// TwinCAT 3 PLC project Sorting_Machine_PLC
// ProgramVersion: 3.1.4024.0
// libraries:
//   Tc2_MC2, * (Beckhoff Automation GmbH)
//   Tc2_Standard, * (Beckhoff Automation GmbH)
//   Tc2_System, * (Beckhoff Automation GmbH)
//   Tc3_Module, * (Beckhoff Automation GmbH)
// project tree:
//   00_Internal PackML/DUTs/ E_PMLState.TcDUT, E_PMLUnitMode.TcDUT
//   00_Internal PackML/POUs/ PS_PackML_StateMachine_Auto.TcPOU, PS_PackML_StateMachine_Maintenance.TcPOU, PS_PackML_StateMachine_Manual.TcPOU, PS_PackML_StateMachine_SemiAuto.TcPOU, PS_PackML_UnitModeManager.TcPOU
//   01_Submodules/Axis/ FB_Axis.TcPOU
//   01_Submodules/Cylinder/ FB_CylinderDiag.TcPOU, FB_CylinderTemp.TcPOU, FB_CylinderTempDiag.TcPOU, FB_CylinderTempRecord.TcPOU, I_Cylinder.TcIO, FB_CylinderBase.TcPOU
//   01_Submodules/Sensor %28signal handling%29/ FB_SignalHandling.TcPOU (not stored), FB_SignalHandlingIntern.TcPOU (not stored), I_SignalHandling.TcIO (not stored), FB_SignalHandlingDelay.TcPOU (not stored)
//   02_Subsystems/ E_StateSeparatingAutoClampBarrier.TcDUT, E_StateSortingAutoAxis.TcDUT, E_StateSortingAutoCylinder.TcDUT, FB_SeparatingModule.TcPOU, FB_SortingModule.TcPOU, FB_SubsystemRoot.TcPOU
//   03_Machine/ FB_Machine.TcPOU
//   / PlcTask.TcTTO
//   04_Application/ MAIN.TcPOU
// real-time tasks:
//   TASK PlcTask: cycle T#10ms, priority 20, ADS port 350

CONFIGURATION Sorting_Machine_PLC
    RESOURCE PLC ON TwinCAT3
        TASK PlcTask(INTERVAL := T#10ms, PRIORITY := 20);
        PROGRAM MAIN WITH PlcTask : MAIN;
    END_RESOURCE
END_CONFIGURATION

// ---- 00_Internal PackML/DUTs/E_PMLState.TcDUT
{attribute 'qualified_only'}
{attribute 'strict'}
TYPE E_PMLState :
(
	UNDEFINED 			:=	0,
	CLEARING			:=	1,
	STOPPED				:=	2,
	STARTING			:=	3,
	IDLE				:=	4,
	SUSPENDED			:=	5,
	EXECUTE				:=	6,
	STOPPING			:=	7,
	ABORTING			:=	8,
	ABORTED				:=	9,
	HOLDING				:=	10,
	HELD				:=	11,
	UNHOLDING			:=	12,
	SUSPENDING			:=	13,
	UNSUSPENDING		:=	14,
	RESETTING			:=	15,
	COMPLETING			:=	16,
	COMPLETE			:=	17
);
END_TYPE

// ---- 00_Internal PackML/DUTs/E_PMLUnitMode.TcDUT
{attribute 'qualified_only'}
{attribute 'strict'}
TYPE E_PMLUnitMode :
(
	UNDEFINED 			:=	0,
	AUTOMATIC			:=	1,
	MAINTENANCE			:=	2,
	MANUAL				:=	3,
	SEMIAUTOMATIC		:=	4,
	DRYRUN				:=	5,
	USERMODE1			:=	6,
	USERMODE2			:=	7,
	IDLE				:=	8,
	ESTOP				:=	9
);
END_TYPE

// ---- 02_Subsystems/E_StateSeparatingAutoClampBarrier.TcDUT
{attribute 'qualified_only'}
{attribute 'strict'}
TYPE E_StateSeparatingAutoClampBarrier :
(
	Init 			:= 0,
	Start,
	CloseClamp,
	OpenBarrier,
	CloseBarrier,
	OpenClamp
);
END_TYPE

// ---- 02_Subsystems/E_StateSortingAutoAxis.TcDUT
{attribute 'qualified_only'}
{attribute 'strict'}
TYPE E_StateSortingAutoAxis :
(
	WaitForCylinderAtWorkPos 			:= 0,
	MoveAxis,
	StopAxis
);
END_TYPE

// ---- 02_Subsystems/E_StateSortingAutoCylinder.TcDUT
{attribute 'qualified_only'}
{attribute 'strict'}
TYPE E_StateSortingAutoCylinder :
(
	BoxDetected 			:= 0,
	MoveCylToWorkPos,
	MoveCylToBasePos
);
END_TYPE

// ---- 01_Submodules/Cylinder/I_Cylinder.TcIO
INTERFACE I_Cylinder

PROPERTY bState_AtBasePos : BOOL
GET
END_GET
END_PROPERTY

PROPERTY bState_AtWorkPos : BOOL
GET
END_GET
END_PROPERTY

PROPERTY bState_MoveToWork : BOOL
GET
END_GET
END_PROPERTY

METHOD MoveToBase
VAR_INPUT
END_VAR
END_METHOD

METHOD MoveToWork
VAR_INPUT
END_VAR
END_METHOD

METHOD Reset
VAR_INPUT
END_VAR
END_METHOD

END_INTERFACE

// ---- 04_Application/MAIN.TcPOU
PROGRAM MAIN
VAR
END_VAR

END_PROGRAM

// ---- 00_Internal PackML/POUs/PS_PackML_StateMachine_Auto.TcPOU
FUNCTION_BLOCK PS_PackML_StateMachine_Auto
VAR_INPUT
	Start					:	BOOL;
	Hold					:	BOOL;
	UnHold					:	BOOL;
	Suspend					:	BOOL;
	UnSuspend				:	BOOL;
	Abort					:	BOOL;
	Stop					:	BOOL;
	Complete				:	BOOL;
	Clear					:	BOOL;
	Reset					:	BOOL;
	StateComplete			:	BOOL;
END_VAR
VAR_OUTPUT
	Status					:	WORD;
	// Transient states
	ST_Starting				:	BOOL;
	ST_Completing			:	BOOL;
	ST_Resetting			:	BOOL;
	ST_Holding				:	BOOL;
	ST_UnHolding			:	BOOL;
	ST_Suspending			:	BOOL;
	ST_UnSuspending			:	BOOL;
	ST_Clearing				:	BOOL;
	ST_Stopping				:	BOOL;
	ST_Aborting				:	BOOL;
	// Final states
	ST_Execute				:	BOOL;
	ST_Complete				:	BOOL;
	ST_Idle					:	BOOL;
	ST_Held					:	BOOL;
	ST_Suspended			:	BOOL;
	ST_Stopped				:	BOOL;
	ST_Aborted				:	BOOL;
	
	Error					:	BOOL;
	ErrorID					:	DWORD;
	ePMLState				:	E_PMLState	:=	E_PMLState.IDLE;
END_VAR
VAR
	ePMLStatePrev			:	E_PMLState;
	bStateChange			:	BOOL;
	bStateCompletePrev		:	BOOL;
END_VAR

	// Check for E_PMLState change
	IF ePMLStatePrev <> ePMLState THEN
		ePMLStatePrev	:=	ePMLState;
		bStateChange	:=	TRUE;
	ELSE
		bStateChange	:=	FALSE;
	END_IF
	
	// change to new state if requested
	CASE ePMLState OF
		E_PMLState.UNDEFINED:
			IF bStateChange	THEN
				ST_Starting				:=	FALSE;
				ST_Completing			:=	FALSE;
				ST_Resetting			:=	FALSE;
				ST_Holding				:=	FALSE;
				ST_UnHolding			:=	FALSE;
				ST_Suspending			:=	FALSE;
				ST_UnSuspending			:=	FALSE;
				ST_Clearing				:=	FALSE;
				ST_Stopping				:=	FALSE;
				ST_Aborting				:=	FALSE;
				
				ST_Execute				:=	FALSE;
				ST_Complete				:=	FALSE;
				ST_Idle					:=	FALSE;
				ST_Held					:=	FALSE;
				ST_Suspended			:=	FALSE;
				ST_Stopped				:=	FALSE;
				ST_Aborted				:=	FALSE;
			END_IF
			
			IF Abort THEN
				ePMLState				:=	E_PMLState.ABORTING;
				ST_Aborting				:=	TRUE;
			ELSIF Stop THEN
				ePMLState				:=	E_PMLState.STOPPING;
				ST_Stopping				:=	TRUE;				
			END_IF
		
		E_PMLState.IDLE:
			IF bStateChange	THEN
				ST_Starting				:=	FALSE;
				ST_Completing			:=	FALSE;
				ST_Resetting			:=	FALSE;
				ST_Holding				:=	FALSE;
				ST_UnHolding			:=	FALSE;
				ST_Suspending			:=	FALSE;
				ST_UnSuspending			:=	FALSE;
				ST_Clearing				:=	FALSE;
				ST_Stopping				:=	FALSE;
				ST_Aborting				:=	FALSE;
				
				ST_Execute				:=	FALSE;
				ST_Complete				:=	FALSE;
				ST_Idle					:=	TRUE;
				ST_Held					:=	FALSE;
				ST_Suspended			:=	FALSE;
				ST_Stopped				:=	FALSE;
				ST_Aborted				:=	FALSE;
			END_IF
			
			IF Abort THEN
				ePMLState				:=	E_PMLState.ABORTING;
				ST_IDLE					:=	FALSE;
				ST_Aborting				:=	TRUE;
			ELSIF Stop THEN
				ePMLState				:=	E_PMLState.STOPPING;
				ST_IDLE					:=	FALSE;
				ST_Stopping				:=	TRUE;
			ELSIF Start THEN
				ePMLState				:=	E_PMLState.STARTING;
				ST_IDLE					:=	FALSE;
				ST_Starting				:=	TRUE;								
			END_IF

		E_PMLState.STARTING:
			IF bStateChange	THEN
				ST_Starting				:=	TRUE;
				ST_Completing			:=	FALSE;
				ST_Resetting			:=	FALSE;
				ST_Holding				:=	FALSE;
				ST_UnHolding			:=	FALSE;
				ST_Suspending			:=	FALSE;
				ST_UnSuspending			:=	FALSE;
				ST_Clearing				:=	FALSE;
				ST_Stopping				:=	FALSE;
				ST_Aborting				:=	FALSE;
				
				ST_Execute				:=	FALSE;
				ST_Complete				:=	FALSE;
				ST_Idle					:=	FALSE;
				ST_Held					:=	FALSE;
				ST_Suspended			:=	FALSE;
				ST_Stopped				:=	FALSE;
				ST_Aborted				:=	FALSE;
			END_IF
			
			IF Abort THEN
				ePMLState				:=	E_PMLState.ABORTING;
				ST_Starting				:=	FALSE;
				ST_Aborting				:=	TRUE;
			ELSIF Stop THEN
				ePMLState				:=	E_PMLState.STOPPING;
				ST_Starting				:=	FALSE;
				ST_Stopping				:=	TRUE;
			ELSIF StateComplete AND NOT bStateCompletePrev THEN
				ePMLState				:=	E_PMLState.EXECUTE;
				bStateCompletePrev		:=	StateComplete;
				ST_Starting				:=	FALSE;
				ST_Execute				:=	TRUE;								
			END_IF

		E_PMLState.EXECUTE:
			IF bStateChange	THEN
				ST_Starting				:=	FALSE;
				ST_Completing			:=	FALSE;
				ST_Resetting			:=	FALSE;
				ST_Holding				:=	FALSE;
				ST_UnHolding			:=	FALSE;
				ST_Suspending			:=	FALSE;
				ST_UnSuspending			:=	FALSE;
				ST_Clearing				:=	FALSE;
				ST_Stopping				:=	FALSE;
				ST_Aborting				:=	FALSE;
				
				ST_Execute				:=	TRUE;
				ST_Complete				:=	FALSE;
				ST_Idle					:=	FALSE;
				ST_Held					:=	FALSE;
				ST_Suspended			:=	FALSE;
				ST_Stopped				:=	FALSE;
				ST_Aborted				:=	FALSE;
			END_IF
			
			IF Abort THEN
				ePMLState				:=	E_PMLState.ABORTING;
				ST_Execute				:=	FALSE;
				ST_Aborting				:=	TRUE;
			ELSIF Stop THEN
				ePMLState				:=	E_PMLState.STOPPING;
				ST_Execute				:=	FALSE;
				ST_Stopping				:=	TRUE;
			ELSIF Hold THEN
				ePMLState				:=	E_PMLState.HOLDING;
				ST_Execute				:=	FALSE;
				ST_Holding				:=	TRUE;
			ELSIF Suspend THEN
				ePMLState				:=	E_PMLState.SUSPENDING;
				ST_Execute				:=	FALSE;
				ST_Suspending			:=	TRUE;
			ELSIF Complete THEN
				ePMLState				:=	E_PMLState.COMPLETING;
				ST_Execute				:=	FALSE;
				ST_Completing			:=	TRUE;	
			END_IF

		E_PMLState.COMPLETING:
			IF bStateChange	THEN
				ST_Starting				:=	FALSE;
				ST_Completing			:=	TRUE;
				ST_Resetting			:=	FALSE;
				ST_Holding				:=	FALSE;
				ST_UnHolding			:=	FALSE;
				ST_Suspending			:=	FALSE;
				ST_UnSuspending			:=	FALSE;
				ST_Clearing				:=	FALSE;
				ST_Stopping				:=	FALSE;
				ST_Aborting				:=	FALSE;
				
				ST_Execute				:=	FALSE;
				ST_Complete				:=	FALSE;
				ST_Idle					:=	FALSE;
				ST_Held					:=	FALSE;
				ST_Suspended			:=	FALSE;
				ST_Stopped				:=	FALSE;
				ST_Aborted				:=	FALSE;
			END_IF
			
			IF Abort THEN
				ePMLState				:=	E_PMLState.ABORTING;
				ST_Completing			:=	FALSE;
				ST_Aborting				:=	TRUE;
			ELSIF Stop THEN
				ePMLState				:=	E_PMLState.STOPPING;
				ST_Completing			:=	FALSE;
				ST_Stopping				:=	TRUE;
			ELSIF StateComplete AND NOT bStateCompletePrev THEN
				ePMLState				:=	E_PMLState.COMPLETE;
				bStateCompletePrev		:=	StateComplete;
				ST_Completing			:=	FALSE;
				ST_Complete				:=	TRUE;								
			END_IF
			
		E_PMLState.COMPLETE:
			IF bStateChange	THEN
				ST_Starting				:=	FALSE;
				ST_Completing			:=	FALSE;
				ST_Resetting			:=	FALSE;
				ST_Holding				:=	FALSE;
				ST_UnHolding			:=	FALSE;
				ST_Suspending			:=	FALSE;
				ST_UnSuspending			:=	FALSE;
				ST_Clearing				:=	FALSE;
				ST_Stopping				:=	FALSE;
				ST_Aborting				:=	FALSE;
				
				ST_Execute				:=	FALSE;
				ST_Complete				:=	TRUE;
				ST_Idle					:=	FALSE;
				ST_Held					:=	FALSE;
				ST_Suspended			:=	FALSE;
				ST_Stopped				:=	FALSE;
				ST_Aborted				:=	FALSE;
			END_IF
			
			IF Abort THEN
				ePMLState				:=	E_PMLState.ABORTING;
				ST_Complete				:=	FALSE;
				ST_Aborting				:=	TRUE;
			ELSIF Stop THEN
				ePMLState				:=	E_PMLState.STOPPING;
				ST_Complete				:=	FALSE;
				ST_Stopping				:=	TRUE;
			ELSIF Reset THEN
				ePMLState				:=	E_PMLState.RESETTING;
				ST_Complete				:=	FALSE;
				ST_Resetting			:=	TRUE;
			END_IF

		E_PMLState.RESETTING:
			IF bStateChange	THEN
				ST_Starting				:=	FALSE;
				ST_Completing			:=	FALSE;
				ST_Resetting			:=	TRUE;
				ST_Holding				:=	FALSE;
				ST_UnHolding			:=	FALSE;
				ST_Suspending			:=	FALSE;
				ST_UnSuspending			:=	FALSE;
				ST_Clearing				:=	FALSE;
				ST_Stopping				:=	FALSE;
				ST_Aborting				:=	FALSE;
				
				ST_Execute				:=	FALSE;
				ST_Complete				:=	FALSE;
				ST_Idle					:=	FALSE;
				ST_Held					:=	FALSE;
				ST_Suspended			:=	FALSE;
				ST_Stopped				:=	FALSE;
				ST_Aborted				:=	FALSE;
			END_IF
			
			IF Abort THEN
				ePMLState				:=	E_PMLState.ABORTING;
				ST_Resetting			:=	FALSE;
				ST_Aborting				:=	TRUE;
			ELSIF Stop THEN
				ePMLState				:=	E_PMLState.STOPPING;
				ST_Resetting			:=	FALSE;
				ST_Stopping				:=	TRUE;
			ELSIF StateComplete AND NOT bStateCompletePrev THEN
				ePMLState				:=	E_PMLState.IDLE;
				bStateCompletePrev		:=	StateComplete;
				ST_Resetting			:=	FALSE;
				ST_Idle					:=	TRUE;								
			END_IF
		
		E_PMLState.HOLDING:
			IF bStateChange	THEN
				ST_Starting				:=	FALSE;
				ST_Completing			:=	FALSE;
				ST_Resetting			:=	FALSE;
				ST_Holding				:=	TRUE;
				ST_UnHolding			:=	FALSE;
				ST_Suspending			:=	FALSE;
				ST_UnSuspending			:=	FALSE;
				ST_Clearing				:=	FALSE;
				ST_Stopping				:=	FALSE;
				ST_Aborting				:=	FALSE;
				
				ST_Execute				:=	FALSE;
				ST_Complete				:=	FALSE;
				ST_Idle					:=	FALSE;
				ST_Held					:=	FALSE;
				ST_Suspended			:=	FALSE;
				ST_Stopped				:=	FALSE;
				ST_Aborted				:=	FALSE;
			END_IF
			
			IF Abort THEN
				ePMLState				:=	E_PMLState.ABORTING;
				ST_Holding				:=	FALSE;
				ST_Aborting				:=	TRUE;
			ELSIF Stop THEN
				ePMLState				:=	E_PMLState.STOPPING;
				ST_Holding				:=	FALSE;
				ST_Stopping				:=	TRUE;
			ELSIF StateComplete AND NOT bStateCompletePrev THEN
				ePMLState				:=	E_PMLState.HELD;
				bStateCompletePrev		:=	StateComplete;
				ST_Holding				:=	FALSE;
				ST_Held					:=	TRUE;								
			END_IF
			
		E_PMLState.HELD:
			IF bStateChange	THEN
				ST_Starting				:=	FALSE;
				ST_Completing			:=	FALSE;
				ST_Resetting			:=	FALSE;
				ST_Holding				:=	FALSE;
				ST_UnHolding			:=	FALSE;
				ST_Suspending			:=	FALSE;
				ST_UnSuspending			:=	FALSE;
				ST_Clearing				:=	FALSE;
				ST_Stopping				:=	FALSE;
				ST_Aborting				:=	FALSE;
				
				ST_Execute				:=	FALSE;
				ST_Complete				:=	FALSE;
				ST_Idle					:=	FALSE;
				ST_Held					:=	TRUE;
				ST_Suspended			:=	FALSE;
				ST_Stopped				:=	FALSE;
				ST_Aborted				:=	FALSE;
			END_IF
			
			IF Abort THEN
				ePMLState				:=	E_PMLState.ABORTING;
				ST_Held					:=	FALSE;
				ST_Aborting				:=	TRUE;
			ELSIF Stop THEN
				ePMLState				:=	E_PMLState.STOPPING;
				ST_Held					:=	FALSE;
				ST_Stopping				:=	TRUE;
			ELSIF UnHold THEN
				ePMLState				:=	E_PMLState.UNHOLDING;
				ST_Held					:=	FALSE;
				ST_UnHolding			:=	TRUE;
			END_IF

		E_PMLState.UNHOLDING:	
			IF bStateChange	THEN
				ST_Starting				:=	FALSE;
				ST_Completing			:=	FALSE;
				ST_Resetting			:=	FALSE;
				ST_Holding				:=	FALSE;
				ST_UnHolding			:=	TRUE;
				ST_Suspending			:=	FALSE;
				ST_UnSuspending			:=	FALSE;
				ST_Clearing				:=	FALSE;
				ST_Stopping				:=	FALSE;
				ST_Aborting				:=	FALSE;
				
				ST_Execute				:=	FALSE;
				ST_Complete				:=	FALSE;
				ST_Idle					:=	FALSE;
				ST_Held					:=	FALSE;
				ST_Suspended			:=	FALSE;
				ST_Stopped				:=	FALSE;
				ST_Aborted				:=	FALSE;
			END_IF
			
			IF Abort THEN
				ePMLState				:=	E_PMLState.ABORTING;
				ST_UnHolding			:=	FALSE;
				ST_Aborting				:=	TRUE;
			ELSIF Stop THEN
				ePMLState				:=	E_PMLState.STOPPING;
				ST_UnHolding			:=	FALSE;
				ST_Stopping				:=	TRUE;
			ELSIF StateComplete AND NOT bStateCompletePrev THEN
				ePMLState				:=	E_PMLState.EXECUTE;
				bStateCompletePrev		:=	StateComplete;
				ST_UnHolding			:=	FALSE;
				ST_Execute				:=	TRUE;								
			END_IF
			
		E_PMLState.SUSPENDING:
			IF bStateChange	THEN
				ST_Starting				:=	FALSE;
				ST_Completing			:=	FALSE;
				ST_Resetting			:=	FALSE;
				ST_Holding				:=	FALSE;
				ST_UnHolding			:=	FALSE;
				ST_Suspending			:=	TRUE;
				ST_UnSuspending			:=	FALSE;
				ST_Clearing				:=	FALSE;
				ST_Stopping				:=	FALSE;
				ST_Aborting				:=	FALSE;
				
				ST_Execute				:=	FALSE;
				ST_Complete				:=	FALSE;
				ST_Idle					:=	FALSE;
				ST_Held					:=	FALSE;
				ST_Suspended			:=	FALSE;
				ST_Stopped				:=	FALSE;
				ST_Aborted				:=	FALSE;
			END_IF
			
			IF Abort THEN
				ePMLState				:=	E_PMLState.ABORTING;
				ST_Suspending			:=	FALSE;
				ST_Aborting				:=	TRUE;
			ELSIF Stop THEN
				ePMLState				:=	E_PMLState.STOPPING;
				ST_Suspending			:=	FALSE;
				ST_Stopping				:=	TRUE;
			ELSIF StateComplete AND NOT bStateCompletePrev THEN
				ePMLState				:=	E_PMLState.SUSPENDED;
				bStateCompletePrev		:=	StateComplete;
				ST_Suspending			:=	FALSE;
				ST_Suspended			:=	TRUE;								
			END_IF
		
		E_PMLState.SUSPENDED:
			IF bStateChange	THEN
				ST_Starting				:=	FALSE;
				ST_Completing			:=	FALSE;
				ST_Resetting			:=	FALSE;
				ST_Holding				:=	FALSE;
				ST_UnHolding			:=	FALSE;
				ST_Suspending			:=	FALSE;
				ST_UnSuspending			:=	FALSE;
				ST_Clearing				:=	FALSE;
				ST_Stopping				:=	FALSE;
				ST_Aborting				:=	FALSE;
				
				ST_Execute				:=	FALSE;
				ST_Complete				:=	FALSE;
				ST_Idle					:=	FALSE;
				ST_Held					:=	FALSE;
				ST_Suspended			:=	TRUE;
				ST_Stopped				:=	FALSE;
				ST_Aborted				:=	FALSE;
			END_IF
			
			IF Abort THEN
				ePMLState				:=	E_PMLState.ABORTING;
				ST_Suspended			:=	FALSE;
				ST_Aborting				:=	TRUE;
			ELSIF Stop THEN
				ePMLState				:=	E_PMLState.STOPPING;
				ST_Suspended			:=	FALSE;
				ST_Stopping				:=	TRUE;
			ELSIF UnSuspend THEN
				ePMLState				:=	E_PMLState.UNSUSPENDING;
				ST_Suspended			:=	FALSE;
				ST_UnSuspending			:=	TRUE;
			END_IF

		E_PMLState.UNSUSPENDING:	
			IF bStateChange	THEN
				ST_Starting				:=	FALSE;
				ST_Completing			:=	FALSE;
				ST_Resetting			:=	FALSE;
				ST_Holding				:=	FALSE;
				ST_UnHolding			:=	FALSE;
				ST_Suspending			:=	FALSE;
				ST_UnSuspending			:=	TRUE;
				ST_Clearing				:=	FALSE;
				ST_Stopping				:=	FALSE;
				ST_Aborting				:=	FALSE;
				
				ST_Execute				:=	FALSE;
				ST_Complete				:=	FALSE;
				ST_Idle					:=	FALSE;
				ST_Held					:=	FALSE;
				ST_Suspended			:=	FALSE;
				ST_Stopped				:=	FALSE;
				ST_Aborted				:=	FALSE;
			END_IF
			
			IF Abort THEN
				ePMLState				:=	E_PMLState.ABORTING;
				ST_UnSuspending			:=	FALSE;
				ST_Aborting				:=	TRUE;
			ELSIF Stop THEN
				ePMLState				:=	E_PMLState.STOPPING;
				ST_UnSuspending			:=	FALSE;
				ST_Stopping				:=	TRUE;
			ELSIF StateComplete AND NOT bStateCompletePrev THEN
				ePMLState				:=	E_PMLState.EXECUTE;
				bStateCompletePrev		:=	StateComplete;
				ST_UnSuspending			:=	FALSE;
				ST_Execute				:=	TRUE;								
			END_IF
		
		E_PMLState.STOPPING:
			IF bStateChange	THEN
				ST_Starting				:=	FALSE;
				ST_Completing			:=	FALSE;
				ST_Resetting			:=	FALSE;
				ST_Holding				:=	FALSE;
				ST_UnHolding			:=	FALSE;
				ST_Suspending			:=	FALSE;
				ST_UnSuspending			:=	FALSE;
				ST_Clearing				:=	FALSE;
				ST_Stopping				:=	TRUE;
				ST_Aborting				:=	FALSE;
				
				ST_Execute				:=	FALSE;
				ST_Complete				:=	FALSE;
				ST_Idle					:=	FALSE;
				ST_Held					:=	FALSE;
				ST_Suspended			:=	FALSE;
				ST_Stopped				:=	FALSE;
				ST_Aborted				:=	FALSE;
			END_IF
			
			IF Abort THEN
				ePMLState				:=	E_PMLState.ABORTING;
				ST_Stopping				:=	FALSE;
				ST_Aborting				:=	TRUE;
			ELSIF StateComplete AND NOT bStateCompletePrev THEN
				ePMLState				:=	E_PMLState.STOPPED;
				bStateCompletePrev		:=	StateComplete;
				ST_Stopping				:=	FALSE;
				ST_Stopped				:=	TRUE;								
			END_IF

		E_PMLState.STOPPED:
			IF bStateChange	THEN
				ST_Starting				:=	FALSE;
				ST_Completing			:=	FALSE;
				ST_Resetting			:=	FALSE;
				ST_Holding				:=	FALSE;
				ST_UnHolding			:=	FALSE;
				ST_Suspending			:=	FALSE;
				ST_UnSuspending			:=	FALSE;
				ST_Clearing				:=	FALSE;
				ST_Stopping				:=	FALSE;
				ST_Aborting				:=	FALSE;
				
				ST_Execute				:=	FALSE;
				ST_Complete				:=	FALSE;
				ST_Idle					:=	FALSE;
				ST_Held					:=	FALSE;
				ST_Suspended			:=	FALSE;
				ST_Stopped				:=	TRUE;
				ST_Aborted				:=	FALSE;
			END_IF
			
			IF Abort THEN
				ePMLState				:=	E_PMLState.ABORTING;
				ST_Stopped				:=	FALSE;
				ST_Aborting				:=	TRUE;
			ELSIF Reset THEN
				ePMLState				:=	E_PMLState.RESETTING;
				ST_Stopped				:=	FALSE;
				ST_Resetting			:=	TRUE;
			END_IF
		
		E_PMLState.ABORTING:
			IF bStateChange	THEN
				ST_Starting				:=	FALSE;
				ST_Completing			:=	FALSE;
				ST_Resetting			:=	FALSE;
				ST_Holding				:=	FALSE;
				ST_UnHolding			:=	FALSE;
				ST_Suspending			:=	FALSE;
				ST_UnSuspending			:=	FALSE;
				ST_Clearing				:=	FALSE;
				ST_Stopping				:=	FALSE;
				ST_Aborting				:=	TRUE;
				
				ST_Execute				:=	FALSE;
				ST_Complete				:=	FALSE;
				ST_Idle					:=	FALSE;
				ST_Held					:=	FALSE;
				ST_Suspended			:=	FALSE;
				ST_Stopped				:=	FALSE;
				ST_Aborted				:=	FALSE;
			END_IF
			
			IF StateComplete AND NOT bStateCompletePrev THEN
				ePMLState				:=	E_PMLState.ABORTED;
				bStateCompletePrev		:=	StateComplete;
				ST_Aborting				:=	FALSE;
				ST_Aborted				:=	TRUE;								
			END_IF
			
		E_PMLState.ABORTED:
			IF bStateChange	THEN
				ST_Starting				:=	FALSE;
				ST_Completing			:=	FALSE;
				ST_Resetting			:=	FALSE;
				ST_Holding				:=	FALSE;
				ST_UnHolding			:=	FALSE;
				ST_Suspending			:=	FALSE;
				ST_UnSuspending			:=	FALSE;
				ST_Clearing				:=	FALSE;
				ST_Stopping				:=	FALSE;
				ST_Aborting				:=	FALSE;
				
				ST_Execute				:=	FALSE;
				ST_Complete				:=	FALSE;
				ST_Idle					:=	FALSE;
				ST_Held					:=	FALSE;
				ST_Suspended			:=	FALSE;
				ST_Stopped				:=	FALSE;
				ST_Aborted				:=	TRUE;
			END_IF
			
			IF Clear THEN
				ePMLState				:=	E_PMLState.CLEARING;
				ST_Aborted				:=	FALSE;
				ST_Clearing				:=	TRUE;
			END_IF
		
		E_PMLState.CLEARING:
			IF bStateChange	THEN
				ST_Starting				:=	FALSE;
				ST_Completing			:=	FALSE;
				ST_Resetting			:=	FALSE;
				ST_Holding				:=	FALSE;
				ST_UnHolding			:=	FALSE;
				ST_Suspending			:=	FALSE;
				ST_UnSuspending			:=	FALSE;
				ST_Clearing				:=	TRUE;
				ST_Stopping				:=	FALSE;
				ST_Aborting				:=	FALSE;
				
				ST_Execute				:=	FALSE;
				ST_Complete				:=	FALSE;
				ST_Idle					:=	FALSE;
				ST_Held					:=	FALSE;
				ST_Suspended			:=	FALSE;
				ST_Stopped				:=	FALSE;
				ST_Aborted				:=	FALSE;
			END_IF
			
			IF Abort THEN
				ePMLState				:=	E_PMLState.ABORTING;
				ST_Clearing				:=	FALSE;
				ST_Aborting				:=	TRUE;
			ELSIF Stop THEN
				ePMLState				:=	E_PMLState.STOPPING;
				ST_Clearing				:=	FALSE;
				ST_Stopping				:=	TRUE;
			ELSIF StateComplete AND NOT bStateCompletePrev THEN
				ePMLState				:=	E_PMLState.STOPPED;
				bStateCompletePrev		:=	StateComplete;
				ST_Clearing				:=	FALSE;
				ST_Stopped				:=	TRUE;								
			END_IF
		
	END_CASE
	
	// bStateCompletePrev := bStateCompletePrev AND StateComplete;

END_FUNCTION_BLOCK

// ---- 00_Internal PackML/POUs/PS_PackML_StateMachine_Maintenance.TcPOU
FUNCTION_BLOCK PS_PackML_StateMachine_Maintenance
VAR_INPUT
	Start					:	BOOL;
	Hold					:	BOOL;
	UnHold					:	BOOL;
	Suspend					:	BOOL;
	UnSuspend				:	BOOL;
	Abort					:	BOOL;
	Stop					:	BOOL;
	Complete				:	BOOL;
	Clear					:	BOOL;
	Reset					:	BOOL;
	StateComplete			:	BOOL;
END_VAR
VAR_OUTPUT
	Status					:	WORD;
	// Transient states
	ST_Starting				:	BOOL;
	ST_Completing			:	BOOL;
	ST_Resetting			:	BOOL;
	ST_Holding				:	BOOL;
	ST_UnHolding			:	BOOL;
	ST_Suspending			:	BOOL;
	ST_UnSuspending			:	BOOL;
	ST_Clearing				:	BOOL;
	ST_Stopping				:	BOOL;
	ST_Aborting				:	BOOL;
	// Final states
	ST_Execute				:	BOOL;
	ST_Complete				:	BOOL;
	ST_Idle					:	BOOL;
	ST_Held					:	BOOL;
	ST_Suspended			:	BOOL;
	ST_Stopped				:	BOOL;
	ST_Aborted				:	BOOL;
	
	Error					:	BOOL;
	ErrorID					:	DWORD;
	ePMLState				:	E_PMLState	:=	E_PMLState.IDLE;
END_VAR
VAR
	ePMLStatePrev			:	E_PMLState;
	bStateChange			:	BOOL;
	bStateCompletePrev		:	BOOL;
END_VAR

	// Check for E_PMLState change
	IF ePMLStatePrev <> ePMLState THEN
		ePMLStatePrev	:=	ePMLState;
		bStateChange	:=	TRUE;
	ELSE
		bStateChange	:=	FALSE;
	END_IF
	
	// change to new state if requested
	CASE ePMLState OF
		E_PMLState.UNDEFINED:
			IF bStateChange	THEN
				ST_Starting				:=	FALSE;
				ST_Completing			:=	FALSE;
				ST_Resetting			:=	FALSE;
				ST_Holding				:=	FALSE;
				ST_UnHolding			:=	FALSE;
				ST_Suspending			:=	FALSE;
				ST_UnSuspending			:=	FALSE;
				ST_Clearing				:=	FALSE;
				ST_Stopping				:=	FALSE;
				ST_Aborting				:=	FALSE;
				
				ST_Execute				:=	FALSE;
				ST_Complete				:=	FALSE;
				ST_Idle					:=	FALSE;
				ST_Held					:=	FALSE;
				ST_Suspended			:=	FALSE;
				ST_Stopped				:=	FALSE;
				ST_Aborted				:=	FALSE;
			END_IF
			
			IF Abort THEN
				ePMLState				:=	E_PMLState.ABORTING;
				ST_Aborting				:=	TRUE;
			ELSIF Stop THEN
				ePMLState				:=	E_PMLState.STOPPING;
				ST_Stopping				:=	TRUE;				
			END_IF
			
		E_PMLState.IDLE:
			IF bStateChange	THEN
				ST_Starting				:=	FALSE;
				ST_Completing			:=	FALSE;
				ST_Resetting			:=	FALSE;
				ST_Holding				:=	FALSE;
				ST_UnHolding			:=	FALSE;
				ST_Suspending			:=	FALSE;
				ST_UnSuspending			:=	FALSE;
				ST_Clearing				:=	FALSE;
				ST_Stopping				:=	FALSE;
				ST_Aborting				:=	FALSE;
				
				ST_Execute				:=	FALSE;
				ST_Complete				:=	FALSE;
				ST_Idle					:=	TRUE;
				ST_Held					:=	FALSE;
				ST_Suspended			:=	FALSE;
				ST_Stopped				:=	FALSE;
				ST_Aborted				:=	FALSE;
			END_IF
			
			IF Abort THEN
				ePMLState				:=	E_PMLState.ABORTING;
				ST_IDLE					:=	FALSE;
				ST_Aborting				:=	TRUE;
			ELSIF Stop THEN
				ePMLState				:=	E_PMLState.STOPPING;
				ST_IDLE					:=	FALSE;
				ST_Stopping				:=	TRUE;
			ELSIF Start THEN
				ePMLState				:=	E_PMLState.STARTING;
				ST_IDLE					:=	FALSE;
				ST_Starting				:=	TRUE;								
			END_IF

		E_PMLState.STARTING:
			IF bStateChange	THEN
				ST_Starting				:=	TRUE;
				ST_Completing			:=	FALSE;
				ST_Resetting			:=	FALSE;
				ST_Holding				:=	FALSE;
				ST_UnHolding			:=	FALSE;
				ST_Suspending			:=	FALSE;
				ST_UnSuspending			:=	FALSE;
				ST_Clearing				:=	FALSE;
				ST_Stopping				:=	FALSE;
				ST_Aborting				:=	FALSE;
				
				ST_Execute				:=	FALSE;
				ST_Complete				:=	FALSE;
				ST_Idle					:=	FALSE;
				ST_Held					:=	FALSE;
				ST_Suspended			:=	FALSE;
				ST_Stopped				:=	FALSE;
				ST_Aborted				:=	FALSE;
			END_IF
			
			IF Abort THEN
				ePMLState				:=	E_PMLState.ABORTING;
				ST_Starting				:=	FALSE;
				ST_Aborting				:=	TRUE;
			ELSIF Stop THEN
				ePMLState				:=	E_PMLState.STOPPING;
				ST_Starting				:=	FALSE;
				ST_Stopping				:=	TRUE;
			ELSIF StateComplete AND NOT bStateCompletePrev THEN
				ePMLState				:=	E_PMLState.EXECUTE;
				bStateCompletePrev		:=	StateComplete;
				ST_Starting				:=	FALSE;
				ST_Execute				:=	TRUE;								
			END_IF

		E_PMLState.EXECUTE:
			IF bStateChange	THEN
				ST_Starting				:=	FALSE;
				ST_Completing			:=	FALSE;
				ST_Resetting			:=	FALSE;
				ST_Holding				:=	FALSE;
				ST_UnHolding			:=	FALSE;
				ST_Suspending			:=	FALSE;
				ST_UnSuspending			:=	FALSE;
				ST_Clearing				:=	FALSE;
				ST_Stopping				:=	FALSE;
				ST_Aborting				:=	FALSE;
				
				ST_Execute				:=	TRUE;
				ST_Complete				:=	FALSE;
				ST_Idle					:=	FALSE;
				ST_Held					:=	FALSE;
				ST_Suspended			:=	FALSE;
				ST_Stopped				:=	FALSE;
				ST_Aborted				:=	FALSE;
			END_IF
			
			IF Abort THEN
				ePMLState				:=	E_PMLState.ABORTING;
				ST_Execute				:=	FALSE;
				ST_Aborting				:=	TRUE;
			ELSIF Stop THEN
				ePMLState				:=	E_PMLState.STOPPING;
				ST_Execute				:=	FALSE;
				ST_Stopping				:=	TRUE;
			ELSIF Hold THEN
				ePMLState				:=	E_PMLState.HOLDING;
				ST_Execute				:=	FALSE;
				ST_Holding				:=	TRUE;
			END_IF

		E_PMLState.RESETTING:
			IF bStateChange	THEN
				ST_Starting				:=	FALSE;
				ST_Completing			:=	FALSE;
				ST_Resetting			:=	TRUE;
				ST_Holding				:=	FALSE;
				ST_UnHolding			:=	FALSE;
				ST_Suspending			:=	FALSE;
				ST_UnSuspending			:=	FALSE;
				ST_Clearing				:=	FALSE;
				ST_Stopping				:=	FALSE;
				ST_Aborting				:=	FALSE;
				
				ST_Execute				:=	FALSE;
				ST_Complete				:=	FALSE;
				ST_Idle					:=	FALSE;
				ST_Held					:=	FALSE;
				ST_Suspended			:=	FALSE;
				ST_Stopped				:=	FALSE;
				ST_Aborted				:=	FALSE;
			END_IF
			
			IF Abort THEN
				ePMLState				:=	E_PMLState.ABORTING;
				ST_Resetting			:=	FALSE;
				ST_Aborting				:=	TRUE;
			ELSIF Stop THEN
				ePMLState				:=	E_PMLState.STOPPING;
				ST_Resetting			:=	FALSE;
				ST_Stopping				:=	TRUE;
			ELSIF StateComplete AND NOT bStateCompletePrev THEN
				ePMLState				:=	E_PMLState.IDLE;
				bStateCompletePrev		:=	StateComplete;
				ST_Resetting			:=	FALSE;
				ST_Idle					:=	TRUE;								
			END_IF
		
		E_PMLState.HOLDING:
			IF bStateChange	THEN
				ST_Starting				:=	FALSE;
				ST_Completing			:=	FALSE;
				ST_Resetting			:=	FALSE;
				ST_Holding				:=	TRUE;
				ST_UnHolding			:=	FALSE;
				ST_Suspending			:=	FALSE;
				ST_UnSuspending			:=	FALSE;
				ST_Clearing				:=	FALSE;
				ST_Stopping				:=	FALSE;
				ST_Aborting				:=	FALSE;
				
				ST_Execute				:=	FALSE;
				ST_Complete				:=	FALSE;
				ST_Idle					:=	FALSE;
				ST_Held					:=	FALSE;
				ST_Suspended			:=	FALSE;
				ST_Stopped				:=	FALSE;
				ST_Aborted				:=	FALSE;
			END_IF
			
			IF Abort THEN
				ePMLState				:=	E_PMLState.ABORTING;
				ST_Holding				:=	FALSE;
				ST_Aborting				:=	TRUE;
			ELSIF Stop THEN
				ePMLState				:=	E_PMLState.STOPPING;
				ST_Holding				:=	FALSE;
				ST_Stopping				:=	TRUE;
			ELSIF StateComplete AND NOT bStateCompletePrev THEN
				ePMLState				:=	E_PMLState.HELD;
				bStateCompletePrev		:=	StateComplete;
				ST_Holding				:=	FALSE;
				ST_Held					:=	TRUE;								
			END_IF
			
		E_PMLState.HELD:
			IF bStateChange	THEN
				ST_Starting				:=	FALSE;
				ST_Completing			:=	FALSE;
				ST_Resetting			:=	FALSE;
				ST_Holding				:=	FALSE;
				ST_UnHolding			:=	FALSE;
				ST_Suspending			:=	FALSE;
				ST_UnSuspending			:=	FALSE;
				ST_Clearing				:=	FALSE;
				ST_Stopping				:=	FALSE;
				ST_Aborting				:=	FALSE;
				
				ST_Execute				:=	FALSE;
				ST_Complete				:=	FALSE;
				ST_Idle					:=	FALSE;
				ST_Held					:=	TRUE;
				ST_Suspended			:=	FALSE;
				ST_Stopped				:=	FALSE;
				ST_Aborted				:=	FALSE;
			END_IF
			
			IF Abort THEN
				ePMLState				:=	E_PMLState.ABORTING;
				ST_Held					:=	FALSE;
				ST_Aborting				:=	TRUE;
			ELSIF Stop THEN
				ePMLState				:=	E_PMLState.STOPPING;
				ST_Held					:=	FALSE;
				ST_Stopping				:=	TRUE;
			ELSIF UnHold THEN
				ePMLState				:=	E_PMLState.UNHOLDING;
				ST_Held					:=	FALSE;
				ST_UnHolding			:=	TRUE;
			END_IF

		E_PMLState.UNHOLDING:	
			IF bStateChange	THEN
				ST_Starting				:=	FALSE;
				ST_Completing			:=	FALSE;
				ST_Resetting			:=	FALSE;
				ST_Holding				:=	FALSE;
				ST_UnHolding			:=	TRUE;
				ST_Suspending			:=	FALSE;
				ST_UnSuspending			:=	FALSE;
				ST_Clearing				:=	FALSE;
				ST_Stopping				:=	FALSE;
				ST_Aborting				:=	FALSE;
				
				ST_Execute				:=	FALSE;
				ST_Complete				:=	FALSE;
				ST_Idle					:=	FALSE;
				ST_Held					:=	FALSE;
				ST_Suspended			:=	FALSE;
				ST_Stopped				:=	FALSE;
				ST_Aborted				:=	FALSE;
			END_IF
			
			IF Abort THEN
				ePMLState				:=	E_PMLState.ABORTING;
				ST_UnHolding			:=	FALSE;
				ST_Aborting				:=	TRUE;
			ELSIF Stop THEN
				ePMLState				:=	E_PMLState.STOPPING;
				ST_UnHolding			:=	FALSE;
				ST_Stopping				:=	TRUE;
			ELSIF StateComplete AND NOT bStateCompletePrev THEN
				ePMLState				:=	E_PMLState.EXECUTE;
				bStateCompletePrev		:=	StateComplete;
				ST_UnHolding			:=	FALSE;
				ST_Execute				:=	TRUE;								
			END_IF
				
		E_PMLState.STOPPING:
			IF bStateChange	THEN
				ST_Starting				:=	FALSE;
				ST_Completing			:=	FALSE;
				ST_Resetting			:=	FALSE;
				ST_Holding				:=	FALSE;
				ST_UnHolding			:=	FALSE;
				ST_Suspending			:=	FALSE;
				ST_UnSuspending			:=	FALSE;
				ST_Clearing				:=	FALSE;
				ST_Stopping				:=	TRUE;
				ST_Aborting				:=	FALSE;
				
				ST_Execute				:=	FALSE;
				ST_Complete				:=	FALSE;
				ST_Idle					:=	FALSE;
				ST_Held					:=	FALSE;
				ST_Suspended			:=	FALSE;
				ST_Stopped				:=	FALSE;
				ST_Aborted				:=	FALSE;
			END_IF
			
			IF Abort THEN
				ePMLState				:=	E_PMLState.ABORTING;
				ST_Stopping				:=	FALSE;
				ST_Aborting				:=	TRUE;
			ELSIF StateComplete AND NOT bStateCompletePrev THEN
				ePMLState				:=	E_PMLState.STOPPED;
				bStateCompletePrev		:=	StateComplete;
				ST_Stopping				:=	FALSE;
				ST_Stopped				:=	TRUE;								
			END_IF

		E_PMLState.STOPPED:
			IF bStateChange	THEN
				ST_Starting				:=	FALSE;
				ST_Completing			:=	FALSE;
				ST_Resetting			:=	FALSE;
				ST_Holding				:=	FALSE;
				ST_UnHolding			:=	FALSE;
				ST_Suspending			:=	FALSE;
				ST_UnSuspending			:=	FALSE;
				ST_Clearing				:=	FALSE;
				ST_Stopping				:=	FALSE;
				ST_Aborting				:=	FALSE;
				
				ST_Execute				:=	FALSE;
				ST_Complete				:=	FALSE;
				ST_Idle					:=	FALSE;
				ST_Held					:=	FALSE;
				ST_Suspended			:=	FALSE;
				ST_Stopped				:=	TRUE;
				ST_Aborted				:=	FALSE;
			END_IF
			
			IF Abort THEN
				ePMLState				:=	E_PMLState.ABORTING;
				ST_Stopped				:=	FALSE;
				ST_Aborting				:=	TRUE;
			ELSIF Reset THEN
				ePMLState				:=	E_PMLState.RESETTING;
				ST_Stopped				:=	FALSE;
				ST_Resetting			:=	TRUE;
			END_IF
		
		E_PMLState.ABORTING:
			IF bStateChange	THEN
				ST_Starting				:=	FALSE;
				ST_Completing			:=	FALSE;
				ST_Resetting			:=	FALSE;
				ST_Holding				:=	FALSE;
				ST_UnHolding			:=	FALSE;
				ST_Suspending			:=	FALSE;
				ST_UnSuspending			:=	FALSE;
				ST_Clearing				:=	FALSE;
				ST_Stopping				:=	FALSE;
				ST_Aborting				:=	TRUE;
				
				ST_Execute				:=	FALSE;
				ST_Complete				:=	FALSE;
				ST_Idle					:=	FALSE;
				ST_Held					:=	FALSE;
				ST_Suspended			:=	FALSE;
				ST_Stopped				:=	FALSE;
				ST_Aborted				:=	FALSE;
			END_IF
			
			IF StateComplete AND NOT bStateCompletePrev THEN
				ePMLState				:=	E_PMLState.ABORTED;
				bStateCompletePrev		:=	StateComplete;
				ST_Aborting				:=	FALSE;
				ST_Aborted				:=	TRUE;								
			END_IF
			
		E_PMLState.ABORTED:
			IF bStateChange	THEN
				ST_Starting				:=	FALSE;
				ST_Completing			:=	FALSE;
				ST_Resetting			:=	FALSE;
				ST_Holding				:=	FALSE;
				ST_UnHolding			:=	FALSE;
				ST_Suspending			:=	FALSE;
				ST_UnSuspending			:=	FALSE;
				ST_Clearing				:=	FALSE;
				ST_Stopping				:=	FALSE;
				ST_Aborting				:=	FALSE;
				
				ST_Execute				:=	FALSE;
				ST_Complete				:=	FALSE;
				ST_Idle					:=	FALSE;
				ST_Held					:=	FALSE;
				ST_Suspended			:=	FALSE;
				ST_Stopped				:=	FALSE;
				ST_Aborted				:=	TRUE;
			END_IF
			
			IF Clear THEN
				ePMLState				:=	E_PMLState.CLEARING;
				ST_Aborted				:=	FALSE;
				ST_Clearing				:=	TRUE;
			END_IF
		
		E_PMLState.CLEARING:
			IF bStateChange	THEN
				ST_Starting				:=	FALSE;
				ST_Completing			:=	FALSE;
				ST_Resetting			:=	FALSE;
				ST_Holding				:=	FALSE;
				ST_UnHolding			:=	FALSE;
				ST_Suspending			:=	FALSE;
				ST_UnSuspending			:=	FALSE;
				ST_Clearing				:=	TRUE;
				ST_Stopping				:=	FALSE;
				ST_Aborting				:=	FALSE;
				
				ST_Execute				:=	FALSE;
				ST_Complete				:=	FALSE;
				ST_Idle					:=	FALSE;
				ST_Held					:=	FALSE;
				ST_Suspended			:=	FALSE;
				ST_Stopped				:=	FALSE;
				ST_Aborted				:=	FALSE;
			END_IF
			
			IF Abort THEN
				ePMLState				:=	E_PMLState.ABORTING;
				ST_Clearing				:=	FALSE;
				ST_Aborting				:=	TRUE;
			ELSIF Stop THEN
				ePMLState				:=	E_PMLState.STOPPING;
				ST_Clearing				:=	FALSE;
				ST_Stopping				:=	TRUE;
			ELSIF StateComplete AND NOT bStateCompletePrev THEN
				ePMLState				:=	E_PMLState.STOPPED;
				bStateCompletePrev		:=	StateComplete;
				ST_Clearing				:=	FALSE;
				ST_Stopped				:=	TRUE;								
			END_IF
		
	END_CASE
	
	// bStateCompletePrev := bStateCompletePrev AND StateComplete;

END_FUNCTION_BLOCK

// ---- 00_Internal PackML/POUs/PS_PackML_StateMachine_Manual.TcPOU
FUNCTION_BLOCK PS_PackML_StateMachine_Manual
VAR_INPUT
	Start					:	BOOL;
	Hold					:	BOOL;
	UnHold					:	BOOL;
	Suspend					:	BOOL;
	UnSuspend				:	BOOL;
	Abort					:	BOOL;
	Stop					:	BOOL;
	Complete				:	BOOL;
	Clear					:	BOOL;
	Reset					:	BOOL;
	StateComplete			:	BOOL;
END_VAR
VAR_OUTPUT
	Status					:	WORD;
	// Transient states
	ST_Starting				:	BOOL;
	ST_Completing			:	BOOL;
	ST_Resetting			:	BOOL;
	ST_Holding				:	BOOL;
	ST_UnHolding			:	BOOL;
	ST_Suspending			:	BOOL;
	ST_UnSuspending			:	BOOL;
	ST_Clearing				:	BOOL;
	ST_Stopping				:	BOOL;
	ST_Aborting				:	BOOL;
	// Final states
	ST_Execute				:	BOOL;
	ST_Complete				:	BOOL;
	ST_Idle					:	BOOL;
	ST_Held					:	BOOL;
	ST_Suspended			:	BOOL;
	ST_Stopped				:	BOOL;
	ST_Aborted				:	BOOL;
	
	Error					:	BOOL;
	ErrorID					:	DWORD;
	ePMLState				:	E_PMLState	:=	E_PMLState.IDLE;
END_VAR
VAR
	ePMLStatePrev			:	E_PMLState;
	bStateChange			:	BOOL;
	bStateCompletePrev		:	BOOL;
END_VAR

	// Check for E_PMLState change
	IF ePMLStatePrev <> ePMLState THEN
		ePMLStatePrev	:=	ePMLState;
		bStateChange	:=	TRUE;
	ELSE
		bStateChange	:=	FALSE;
	END_IF
	
	// change to new state if requested
	CASE ePMLState OF
		E_PMLState.UNDEFINED:
			IF bStateChange	THEN
				ST_Starting				:=	FALSE;
				ST_Completing			:=	FALSE;
				ST_Resetting			:=	FALSE;
				ST_Holding				:=	FALSE;
				ST_UnHolding			:=	FALSE;
				ST_Suspending			:=	FALSE;
				ST_UnSuspending			:=	FALSE;
				ST_Clearing				:=	FALSE;
				ST_Stopping				:=	FALSE;
				ST_Aborting				:=	FALSE;
				
				ST_Execute				:=	FALSE;
				ST_Complete				:=	FALSE;
				ST_Idle					:=	FALSE;
				ST_Held					:=	FALSE;
				ST_Suspended			:=	FALSE;
				ST_Stopped				:=	FALSE;
				ST_Aborted				:=	FALSE;
			END_IF
			
			IF Abort THEN
				ePMLState				:=	E_PMLState.ABORTING;
				ST_Aborting				:=	TRUE;
			ELSIF Stop THEN
				ePMLState				:=	E_PMLState.STOPPING;
				ST_Stopping				:=	TRUE;				
			END_IF
		E_PMLState.IDLE:
			IF bStateChange	THEN
				ST_Starting				:=	FALSE;
				ST_Completing			:=	FALSE;
				ST_Resetting			:=	FALSE;
				ST_Holding				:=	FALSE;
				ST_UnHolding			:=	FALSE;
				ST_Suspending			:=	FALSE;
				ST_UnSuspending			:=	FALSE;
				ST_Clearing				:=	FALSE;
				ST_Stopping				:=	FALSE;
				ST_Aborting				:=	FALSE;
				
				ST_Execute				:=	FALSE;
				ST_Complete				:=	FALSE;
				ST_Idle					:=	TRUE;
				ST_Held					:=	FALSE;
				ST_Suspended			:=	FALSE;
				ST_Stopped				:=	FALSE;
				ST_Aborted				:=	FALSE;
			END_IF
			
			IF Abort THEN
				ePMLState				:=	E_PMLState.ABORTING;
				ST_IDLE					:=	FALSE;
				ST_Aborting				:=	TRUE;
			ELSIF Stop THEN
				ePMLState				:=	E_PMLState.STOPPING;
				ST_IDLE					:=	FALSE;
				ST_Stopping				:=	TRUE;
			ELSIF Start THEN
				ePMLState				:=	E_PMLState.STARTING;
				ST_IDLE					:=	FALSE;
				ST_Starting				:=	TRUE;								
			END_IF

		E_PMLState.STARTING:
			IF bStateChange	THEN
				ST_Starting				:=	TRUE;
				ST_Completing			:=	FALSE;
				ST_Resetting			:=	FALSE;
				ST_Holding				:=	FALSE;
				ST_UnHolding			:=	FALSE;
				ST_Suspending			:=	FALSE;
				ST_UnSuspending			:=	FALSE;
				ST_Clearing				:=	FALSE;
				ST_Stopping				:=	FALSE;
				ST_Aborting				:=	FALSE;
				
				ST_Execute				:=	FALSE;
				ST_Complete				:=	FALSE;
				ST_Idle					:=	FALSE;
				ST_Held					:=	FALSE;
				ST_Suspended			:=	FALSE;
				ST_Stopped				:=	FALSE;
				ST_Aborted				:=	FALSE;
			END_IF
			
			IF Abort THEN
				ePMLState				:=	E_PMLState.ABORTING;
				ST_Starting				:=	FALSE;
				ST_Aborting				:=	TRUE;
			ELSIF Stop THEN
				ePMLState				:=	E_PMLState.STOPPING;
				ST_Starting				:=	FALSE;
				ST_Stopping				:=	TRUE;
			ELSIF StateComplete AND NOT bStateCompletePrev THEN
				ePMLState				:=	E_PMLState.EXECUTE;
				bStateCompletePrev		:=	StateComplete;
				ST_Starting				:=	FALSE;
				ST_Execute				:=	TRUE;								
			END_IF

		E_PMLState.EXECUTE:
			IF bStateChange	THEN
				ST_Starting				:=	FALSE;
				ST_Completing			:=	FALSE;
				ST_Resetting			:=	FALSE;
				ST_Holding				:=	FALSE;
				ST_UnHolding			:=	FALSE;
				ST_Suspending			:=	FALSE;
				ST_UnSuspending			:=	FALSE;
				ST_Clearing				:=	FALSE;
				ST_Stopping				:=	FALSE;
				ST_Aborting				:=	FALSE;
				
				ST_Execute				:=	TRUE;
				ST_Complete				:=	FALSE;
				ST_Idle					:=	FALSE;
				ST_Held					:=	FALSE;
				ST_Suspended			:=	FALSE;
				ST_Stopped				:=	FALSE;
				ST_Aborted				:=	FALSE;
			END_IF
			
			IF Abort THEN
				ePMLState				:=	E_PMLState.ABORTING;
				ST_Execute				:=	FALSE;
				ST_Aborting				:=	TRUE;
			ELSIF Stop THEN
				ePMLState				:=	E_PMLState.STOPPING;
				ST_Execute				:=	FALSE;
				ST_Stopping				:=	TRUE;
			END_IF

		E_PMLState.RESETTING:
			IF bStateChange	THEN
				ST_Starting				:=	FALSE;
				ST_Completing			:=	FALSE;
				ST_Resetting			:=	TRUE;
				ST_Holding				:=	FALSE;
				ST_UnHolding			:=	FALSE;
				ST_Suspending			:=	FALSE;
				ST_UnSuspending			:=	FALSE;
				ST_Clearing				:=	FALSE;
				ST_Stopping				:=	FALSE;
				ST_Aborting				:=	FALSE;
				
				ST_Execute				:=	FALSE;
				ST_Complete				:=	FALSE;
				ST_Idle					:=	FALSE;
				ST_Held					:=	FALSE;
				ST_Suspended			:=	FALSE;
				ST_Stopped				:=	FALSE;
				ST_Aborted				:=	FALSE;
			END_IF
			
			IF Abort THEN
				ePMLState				:=	E_PMLState.ABORTING;
				ST_Resetting			:=	FALSE;
				ST_Aborting				:=	TRUE;
			ELSIF Stop THEN
				ePMLState				:=	E_PMLState.STOPPING;
				ST_Resetting			:=	FALSE;
				ST_Stopping				:=	TRUE;
			ELSIF StateComplete AND NOT bStateCompletePrev THEN
				ePMLState				:=	E_PMLState.IDLE;
				bStateCompletePrev		:=	StateComplete;
				ST_Resetting			:=	FALSE;
				ST_Idle					:=	TRUE;								
			END_IF
		
		E_PMLState.STOPPING:
			IF bStateChange	THEN
				ST_Starting				:=	FALSE;
				ST_Completing			:=	FALSE;
				ST_Resetting			:=	FALSE;
				ST_Holding				:=	FALSE;
				ST_UnHolding			:=	FALSE;
				ST_Suspending			:=	FALSE;
				ST_UnSuspending			:=	FALSE;
				ST_Clearing				:=	FALSE;
				ST_Stopping				:=	TRUE;
				ST_Aborting				:=	FALSE;
				
				ST_Execute				:=	FALSE;
				ST_Complete				:=	FALSE;
				ST_Idle					:=	FALSE;
				ST_Held					:=	FALSE;
				ST_Suspended			:=	FALSE;
				ST_Stopped				:=	FALSE;
				ST_Aborted				:=	FALSE;
			END_IF
			
			IF Abort THEN
				ePMLState				:=	E_PMLState.ABORTING;
				ST_Stopping				:=	FALSE;
				ST_Aborting				:=	TRUE;
			ELSIF StateComplete AND NOT bStateCompletePrev THEN
				ePMLState				:=	E_PMLState.STOPPED;
				bStateCompletePrev		:=	StateComplete;
				ST_Stopping				:=	FALSE;
				ST_Stopped				:=	TRUE;								
			END_IF

		E_PMLState.STOPPED:
			IF bStateChange	THEN
				ST_Starting				:=	FALSE;
				ST_Completing			:=	FALSE;
				ST_Resetting			:=	FALSE;
				ST_Holding				:=	FALSE;
				ST_UnHolding			:=	FALSE;
				ST_Suspending			:=	FALSE;
				ST_UnSuspending			:=	FALSE;
				ST_Clearing				:=	FALSE;
				ST_Stopping				:=	FALSE;
				ST_Aborting				:=	FALSE;
				
				ST_Execute				:=	FALSE;
				ST_Complete				:=	FALSE;
				ST_Idle					:=	FALSE;
				ST_Held					:=	FALSE;
				ST_Suspended			:=	FALSE;
				ST_Stopped				:=	TRUE;
				ST_Aborted				:=	FALSE;
			END_IF
			
			IF Abort THEN
				ePMLState				:=	E_PMLState.ABORTING;
				ST_Stopped				:=	FALSE;
				ST_Aborting				:=	TRUE;
			ELSIF Reset THEN
				ePMLState				:=	E_PMLState.RESETTING;
				ST_Stopped				:=	FALSE;
				ST_Resetting			:=	TRUE;
			END_IF
		
		E_PMLState.ABORTING:
			IF bStateChange	THEN
				ST_Starting				:=	FALSE;
				ST_Completing			:=	FALSE;
				ST_Resetting			:=	FALSE;
				ST_Holding				:=	FALSE;
				ST_UnHolding			:=	FALSE;
				ST_Suspending			:=	FALSE;
				ST_UnSuspending			:=	FALSE;
				ST_Clearing				:=	FALSE;
				ST_Stopping				:=	FALSE;
				ST_Aborting				:=	TRUE;
				
				ST_Execute				:=	FALSE;
				ST_Complete				:=	FALSE;
				ST_Idle					:=	FALSE;
				ST_Held					:=	FALSE;
				ST_Suspended			:=	FALSE;
				ST_Stopped				:=	FALSE;
				ST_Aborted				:=	FALSE;
			END_IF
			
			IF StateComplete AND NOT bStateCompletePrev THEN
				ePMLState				:=	E_PMLState.ABORTED;
				bStateCompletePrev		:=	StateComplete;
				ST_Aborting				:=	FALSE;
				ST_Aborted				:=	TRUE;								
			END_IF
			
		E_PMLState.ABORTED:
			IF bStateChange	THEN
				ST_Starting				:=	FALSE;
				ST_Completing			:=	FALSE;
				ST_Resetting			:=	FALSE;
				ST_Holding				:=	FALSE;
				ST_UnHolding			:=	FALSE;
				ST_Suspending			:=	FALSE;
				ST_UnSuspending			:=	FALSE;
				ST_Clearing				:=	FALSE;
				ST_Stopping				:=	FALSE;
				ST_Aborting				:=	FALSE;
				
				ST_Execute				:=	FALSE;
				ST_Complete				:=	FALSE;
				ST_Idle					:=	FALSE;
				ST_Held					:=	FALSE;
				ST_Suspended			:=	FALSE;
				ST_Stopped				:=	FALSE;
				ST_Aborted				:=	TRUE;
			END_IF
			
			IF Clear THEN
				ePMLState				:=	E_PMLState.CLEARING;
				ST_Aborted				:=	FALSE;
				ST_Clearing				:=	TRUE;
			END_IF
		
		E_PMLState.CLEARING:
			IF bStateChange	THEN
				ST_Starting				:=	FALSE;
				ST_Completing			:=	FALSE;
				ST_Resetting			:=	FALSE;
				ST_Holding				:=	FALSE;
				ST_UnHolding			:=	FALSE;
				ST_Suspending			:=	FALSE;
				ST_UnSuspending			:=	FALSE;
				ST_Clearing				:=	TRUE;
				ST_Stopping				:=	FALSE;
				ST_Aborting				:=	FALSE;
				
				ST_Execute				:=	FALSE;
				ST_Complete				:=	FALSE;
				ST_Idle					:=	FALSE;
				ST_Held					:=	FALSE;
				ST_Suspended			:=	FALSE;
				ST_Stopped				:=	FALSE;
				ST_Aborted				:=	FALSE;
			END_IF
			
			IF Abort THEN
				ePMLState				:=	E_PMLState.ABORTING;
				ST_Clearing				:=	FALSE;
				ST_Aborting				:=	TRUE;
			ELSIF Stop THEN
				ePMLState				:=	E_PMLState.STOPPING;
				ST_Clearing				:=	FALSE;
				ST_Stopping				:=	TRUE;
			ELSIF StateComplete AND NOT bStateCompletePrev THEN
				ePMLState				:=	E_PMLState.STOPPED;
				bStateCompletePrev		:=	StateComplete;
				ST_Clearing				:=	FALSE;
				ST_Stopped				:=	TRUE;								
			END_IF
		
	END_CASE
	
	// bStateCompletePrev := bStateCompletePrev AND StateComplete;

END_FUNCTION_BLOCK

// ---- 00_Internal PackML/POUs/PS_PackML_StateMachine_SemiAuto.TcPOU
FUNCTION_BLOCK PS_PackML_StateMachine_SemiAuto
VAR_INPUT
	Start					:	BOOL;
	Hold					:	BOOL;
	UnHold					:	BOOL;
	Suspend					:	BOOL;
	UnSuspend				:	BOOL;
	Abort					:	BOOL;
	Stop					:	BOOL;
	Complete				:	BOOL;
	Clear					:	BOOL;
	Reset					:	BOOL;
	StateComplete			:	BOOL;
END_VAR
VAR_OUTPUT
	Status					:	WORD;
	// Transient states
	ST_Starting				:	BOOL;
	ST_Completing			:	BOOL;
	ST_Resetting			:	BOOL;
	ST_Holding				:	BOOL;
	ST_UnHolding			:	BOOL;
	ST_Suspending			:	BOOL;
	ST_UnSuspending			:	BOOL;
	ST_Clearing				:	BOOL;
	ST_Stopping				:	BOOL;
	ST_Aborting				:	BOOL;
	// Final states
	ST_Execute				:	BOOL;
	ST_Complete				:	BOOL;
	ST_Idle					:	BOOL;
	ST_Held					:	BOOL;
	ST_Suspended			:	BOOL;
	ST_Stopped				:	BOOL;
	ST_Aborted				:	BOOL;
	
	Error					:	BOOL;
	ErrorID					:	DWORD;
	ePMLState				:	E_PMLState	:=	E_PMLState.IDLE;
END_VAR
VAR
	ePMLStatePrev			:	E_PMLState;
	bStateChange			:	BOOL;
	bStateCompletePrev		:	BOOL;
END_VAR

	// Check for E_PMLState change
	IF ePMLStatePrev <> ePMLState THEN
		ePMLStatePrev	:=	ePMLState;
		bStateChange	:=	TRUE;
	ELSE
		bStateChange	:=	FALSE;
	END_IF
	
	// change to new state if requested
	CASE ePMLState OF
		E_PMLState.UNDEFINED:
			IF bStateChange	THEN
				ST_Starting				:=	FALSE;
				ST_Completing			:=	FALSE;
				ST_Resetting			:=	FALSE;
				ST_Holding				:=	FALSE;
				ST_UnHolding			:=	FALSE;
				ST_Suspending			:=	FALSE;
				ST_UnSuspending			:=	FALSE;
				ST_Clearing				:=	FALSE;
				ST_Stopping				:=	FALSE;
				ST_Aborting				:=	FALSE;
				
				ST_Execute				:=	FALSE;
				ST_Complete				:=	FALSE;
				ST_Idle					:=	FALSE;
				ST_Held					:=	FALSE;
				ST_Suspended			:=	FALSE;
				ST_Stopped				:=	FALSE;
				ST_Aborted				:=	FALSE;
			END_IF
			
			IF Abort THEN
				ePMLState				:=	E_PMLState.ABORTING;
				ST_Aborting				:=	TRUE;
			ELSIF Stop THEN
				ePMLState				:=	E_PMLState.STOPPING;
				ST_Stopping				:=	TRUE;				
			END_IF
		E_PMLState.IDLE:
			IF bStateChange	THEN
				ST_Starting				:=	FALSE;
				ST_Completing			:=	FALSE;
				ST_Resetting			:=	FALSE;
				ST_Holding				:=	FALSE;
				ST_UnHolding			:=	FALSE;
				ST_Suspending			:=	FALSE;
				ST_UnSuspending			:=	FALSE;
				ST_Clearing				:=	FALSE;
				ST_Stopping				:=	FALSE;
				ST_Aborting				:=	FALSE;
				
				ST_Execute				:=	FALSE;
				ST_Complete				:=	FALSE;
				ST_Idle					:=	TRUE;
				ST_Held					:=	FALSE;
				ST_Suspended			:=	FALSE;
				ST_Stopped				:=	FALSE;
				ST_Aborted				:=	FALSE;
			END_IF
			
			IF Abort THEN
				ePMLState				:=	E_PMLState.ABORTING;
				ST_IDLE					:=	FALSE;
				ST_Aborting				:=	TRUE;
			ELSIF Stop THEN
				ePMLState				:=	E_PMLState.STOPPING;
				ST_IDLE					:=	FALSE;
				ST_Stopping				:=	TRUE;
			ELSIF Start THEN
				ePMLState				:=	E_PMLState.STARTING;
				ST_IDLE					:=	FALSE;
				ST_Starting				:=	TRUE;								
			END_IF

		E_PMLState.STARTING:
			IF bStateChange	THEN
				ST_Starting				:=	TRUE;
				ST_Completing			:=	FALSE;
				ST_Resetting			:=	FALSE;
				ST_Holding				:=	FALSE;
				ST_UnHolding			:=	FALSE;
				ST_Suspending			:=	FALSE;
				ST_UnSuspending			:=	FALSE;
				ST_Clearing				:=	FALSE;
				ST_Stopping				:=	FALSE;
				ST_Aborting				:=	FALSE;
				
				ST_Execute				:=	FALSE;
				ST_Complete				:=	FALSE;
				ST_Idle					:=	FALSE;
				ST_Held					:=	FALSE;
				ST_Suspended			:=	FALSE;
				ST_Stopped				:=	FALSE;
				ST_Aborted				:=	FALSE;
			END_IF
			
			IF Abort THEN
				ePMLState				:=	E_PMLState.ABORTING;
				ST_Starting				:=	FALSE;
				ST_Aborting				:=	TRUE;
			ELSIF Stop THEN
				ePMLState				:=	E_PMLState.STOPPING;
				ST_Starting				:=	FALSE;
				ST_Stopping				:=	TRUE;
			ELSIF StateComplete AND NOT bStateCompletePrev THEN
				ePMLState				:=	E_PMLState.EXECUTE;
				bStateCompletePrev		:=	StateComplete;
				ST_Starting				:=	FALSE;
				ST_Execute				:=	TRUE;								
			END_IF

		E_PMLState.EXECUTE:
			IF bStateChange	THEN
				ST_Starting				:=	FALSE;
				ST_Completing			:=	FALSE;
				ST_Resetting			:=	FALSE;
				ST_Holding				:=	FALSE;
				ST_UnHolding			:=	FALSE;
				ST_Suspending			:=	FALSE;
				ST_UnSuspending			:=	FALSE;
				ST_Clearing				:=	FALSE;
				ST_Stopping				:=	FALSE;
				ST_Aborting				:=	FALSE;
				
				ST_Execute				:=	TRUE;
				ST_Complete				:=	FALSE;
				ST_Idle					:=	FALSE;
				ST_Held					:=	FALSE;
				ST_Suspended			:=	FALSE;
				ST_Stopped				:=	FALSE;
				ST_Aborted				:=	FALSE;
			END_IF
			
			IF Abort THEN
				ePMLState				:=	E_PMLState.ABORTING;
				ST_Execute				:=	FALSE;
				ST_Aborting				:=	TRUE;
			ELSIF Stop THEN
				ePMLState				:=	E_PMLState.STOPPING;
				ST_Execute				:=	FALSE;
				ST_Stopping				:=	TRUE;
			ELSIF Hold THEN
				ePMLState				:=	E_PMLState.HOLDING;
				ST_Execute				:=	FALSE;
				ST_Holding				:=	TRUE;
			ELSIF Suspend THEN
				ePMLState				:=	E_PMLState.SUSPENDING;
				ST_Execute				:=	FALSE;
				ST_Suspending			:=	TRUE;
			ELSIF Complete THEN
				ePMLState				:=	E_PMLState.COMPLETING;
				ST_Execute				:=	FALSE;
				ST_Completing			:=	TRUE;	
			END_IF

		E_PMLState.COMPLETING:
			IF bStateChange	THEN
				ST_Starting				:=	FALSE;
				ST_Completing			:=	TRUE;
				ST_Resetting			:=	FALSE;
				ST_Holding				:=	FALSE;
				ST_UnHolding			:=	FALSE;
				ST_Suspending			:=	FALSE;
				ST_UnSuspending			:=	FALSE;
				ST_Clearing				:=	FALSE;
				ST_Stopping				:=	FALSE;
				ST_Aborting				:=	FALSE;
				
				ST_Execute				:=	FALSE;
				ST_Complete				:=	FALSE;
				ST_Idle					:=	FALSE;
				ST_Held					:=	FALSE;
				ST_Suspended			:=	FALSE;
				ST_Stopped				:=	FALSE;
				ST_Aborted				:=	FALSE;
			END_IF
			
			IF Abort THEN
				ePMLState				:=	E_PMLState.ABORTING;
				ST_Completing			:=	FALSE;
				ST_Aborting				:=	TRUE;
			ELSIF Stop THEN
				ePMLState				:=	E_PMLState.STOPPING;
				ST_Completing			:=	FALSE;
				ST_Stopping				:=	TRUE;
			ELSIF StateComplete AND NOT bStateCompletePrev THEN
				ePMLState				:=	E_PMLState.COMPLETE;
				bStateCompletePrev		:=	StateComplete;
				ST_Completing			:=	FALSE;
				ST_Complete				:=	TRUE;								
			END_IF
			
		E_PMLState.COMPLETE:
			IF bStateChange	THEN
				ST_Starting				:=	FALSE;
				ST_Completing			:=	FALSE;
				ST_Resetting			:=	FALSE;
				ST_Holding				:=	FALSE;
				ST_UnHolding			:=	FALSE;
				ST_Suspending			:=	FALSE;
				ST_UnSuspending			:=	FALSE;
				ST_Clearing				:=	FALSE;
				ST_Stopping				:=	FALSE;
				ST_Aborting				:=	FALSE;
				
				ST_Execute				:=	FALSE;
				ST_Complete				:=	TRUE;
				ST_Idle					:=	FALSE;
				ST_Held					:=	FALSE;
				ST_Suspended			:=	FALSE;
				ST_Stopped				:=	FALSE;
				ST_Aborted				:=	FALSE;
			END_IF
			
			IF Abort THEN
				ePMLState				:=	E_PMLState.ABORTING;
				ST_Complete				:=	FALSE;
				ST_Aborting				:=	TRUE;
			ELSIF Stop THEN
				ePMLState				:=	E_PMLState.STOPPING;
				ST_Complete				:=	FALSE;
				ST_Stopping				:=	TRUE;
			ELSIF Reset THEN
				ePMLState				:=	E_PMLState.RESETTING;
				ST_Complete				:=	FALSE;
				ST_Resetting			:=	TRUE;
			END_IF

		E_PMLState.RESETTING:
			IF bStateChange	THEN
				ST_Starting				:=	FALSE;
				ST_Completing			:=	FALSE;
				ST_Resetting			:=	TRUE;
				ST_Holding				:=	FALSE;
				ST_UnHolding			:=	FALSE;
				ST_Suspending			:=	FALSE;
				ST_UnSuspending			:=	FALSE;
				ST_Clearing				:=	FALSE;
				ST_Stopping				:=	FALSE;
				ST_Aborting				:=	FALSE;
				
				ST_Execute				:=	FALSE;
				ST_Complete				:=	FALSE;
				ST_Idle					:=	FALSE;
				ST_Held					:=	FALSE;
				ST_Suspended			:=	FALSE;
				ST_Stopped				:=	FALSE;
				ST_Aborted				:=	FALSE;
			END_IF
			
			IF Abort THEN
				ePMLState				:=	E_PMLState.ABORTING;
				ST_Resetting			:=	FALSE;
				ST_Aborting				:=	TRUE;
			ELSIF Stop THEN
				ePMLState				:=	E_PMLState.STOPPING;
				ST_Resetting			:=	FALSE;
				ST_Stopping				:=	TRUE;
			ELSIF StateComplete AND NOT bStateCompletePrev THEN
				ePMLState				:=	E_PMLState.IDLE;
				bStateCompletePrev		:=	StateComplete;
				ST_Resetting			:=	FALSE;
				ST_Idle					:=	TRUE;								
			END_IF
		
		E_PMLState.HOLDING:
			IF bStateChange	THEN
				ST_Starting				:=	FALSE;
				ST_Completing			:=	FALSE;
				ST_Resetting			:=	FALSE;
				ST_Holding				:=	TRUE;
				ST_UnHolding			:=	FALSE;
				ST_Suspending			:=	FALSE;
				ST_UnSuspending			:=	FALSE;
				ST_Clearing				:=	FALSE;
				ST_Stopping				:=	FALSE;
				ST_Aborting				:=	FALSE;
				
				ST_Execute				:=	FALSE;
				ST_Complete				:=	FALSE;
				ST_Idle					:=	FALSE;
				ST_Held					:=	FALSE;
				ST_Suspended			:=	FALSE;
				ST_Stopped				:=	FALSE;
				ST_Aborted				:=	FALSE;
			END_IF
			
			IF Abort THEN
				ePMLState				:=	E_PMLState.ABORTING;
				ST_Holding				:=	FALSE;
				ST_Aborting				:=	TRUE;
			ELSIF Stop THEN
				ePMLState				:=	E_PMLState.STOPPING;
				ST_Holding				:=	FALSE;
				ST_Stopping				:=	TRUE;
			ELSIF StateComplete AND NOT bStateCompletePrev THEN
				ePMLState				:=	E_PMLState.HELD;
				bStateCompletePrev		:=	StateComplete;
				ST_Holding				:=	FALSE;
				ST_Held					:=	TRUE;								
			END_IF
			
		E_PMLState.HELD:
			IF bStateChange	THEN
				ST_Starting				:=	FALSE;
				ST_Completing			:=	FALSE;
				ST_Resetting			:=	FALSE;
				ST_Holding				:=	FALSE;
				ST_UnHolding			:=	FALSE;
				ST_Suspending			:=	FALSE;
				ST_UnSuspending			:=	FALSE;
				ST_Clearing				:=	FALSE;
				ST_Stopping				:=	FALSE;
				ST_Aborting				:=	FALSE;
				
				ST_Execute				:=	FALSE;
				ST_Complete				:=	FALSE;
				ST_Idle					:=	FALSE;
				ST_Held					:=	TRUE;
				ST_Suspended			:=	FALSE;
				ST_Stopped				:=	FALSE;
				ST_Aborted				:=	FALSE;
			END_IF
			
			IF Abort THEN
				ePMLState				:=	E_PMLState.ABORTING;
				ST_Held					:=	FALSE;
				ST_Aborting				:=	TRUE;
			ELSIF Stop THEN
				ePMLState				:=	E_PMLState.STOPPING;
				ST_Held					:=	FALSE;
				ST_Stopping				:=	TRUE;
			ELSIF UnHold THEN
				ePMLState				:=	E_PMLState.UNHOLDING;
				ST_Held					:=	FALSE;
				ST_UnHolding			:=	TRUE;
			END_IF

		E_PMLState.UNHOLDING:	
			IF bStateChange	THEN
				ST_Starting				:=	FALSE;
				ST_Completing			:=	FALSE;
				ST_Resetting			:=	FALSE;
				ST_Holding				:=	FALSE;
				ST_UnHolding			:=	TRUE;
				ST_Suspending			:=	FALSE;
				ST_UnSuspending			:=	FALSE;
				ST_Clearing				:=	FALSE;
				ST_Stopping				:=	FALSE;
				ST_Aborting				:=	FALSE;
				
				ST_Execute				:=	FALSE;
				ST_Complete				:=	FALSE;
				ST_Idle					:=	FALSE;
				ST_Held					:=	FALSE;
				ST_Suspended			:=	FALSE;
				ST_Stopped				:=	FALSE;
				ST_Aborted				:=	FALSE;
			END_IF
			
			IF Abort THEN
				ePMLState				:=	E_PMLState.ABORTING;
				ST_UnHolding			:=	FALSE;
				ST_Aborting				:=	TRUE;
			ELSIF Stop THEN
				ePMLState				:=	E_PMLState.STOPPING;
				ST_UnHolding			:=	FALSE;
				ST_Stopping				:=	TRUE;
			ELSIF StateComplete AND NOT bStateCompletePrev THEN
				ePMLState				:=	E_PMLState.EXECUTE;
				bStateCompletePrev		:=	StateComplete;
				ST_UnHolding			:=	FALSE;
				ST_Execute				:=	TRUE;								
			END_IF
			
		E_PMLState.SUSPENDING:
			IF bStateChange	THEN
				ST_Starting				:=	FALSE;
				ST_Completing			:=	FALSE;
				ST_Resetting			:=	FALSE;
				ST_Holding				:=	FALSE;
				ST_UnHolding			:=	FALSE;
				ST_Suspending			:=	TRUE;
				ST_UnSuspending			:=	FALSE;
				ST_Clearing				:=	FALSE;
				ST_Stopping				:=	FALSE;
				ST_Aborting				:=	FALSE;
				
				ST_Execute				:=	FALSE;
				ST_Complete				:=	FALSE;
				ST_Idle					:=	FALSE;
				ST_Held					:=	FALSE;
				ST_Suspended			:=	FALSE;
				ST_Stopped				:=	FALSE;
				ST_Aborted				:=	FALSE;
			END_IF
			
			IF Abort THEN
				ePMLState				:=	E_PMLState.ABORTING;
				ST_Suspending			:=	FALSE;
				ST_Aborting				:=	TRUE;
			ELSIF Stop THEN
				ePMLState				:=	E_PMLState.STOPPING;
				ST_Suspending			:=	FALSE;
				ST_Stopping				:=	TRUE;
			ELSIF StateComplete AND NOT bStateCompletePrev THEN
				ePMLState				:=	E_PMLState.SUSPENDED;
				bStateCompletePrev		:=	StateComplete;
				ST_Suspending			:=	FALSE;
				ST_Suspended			:=	TRUE;								
			END_IF
		
		E_PMLState.SUSPENDED:
			IF bStateChange	THEN
				ST_Starting				:=	FALSE;
				ST_Completing			:=	FALSE;
				ST_Resetting			:=	FALSE;
				ST_Holding				:=	FALSE;
				ST_UnHolding			:=	FALSE;
				ST_Suspending			:=	FALSE;
				ST_UnSuspending			:=	FALSE;
				ST_Clearing				:=	FALSE;
				ST_Stopping				:=	FALSE;
				ST_Aborting				:=	FALSE;
				
				ST_Execute				:=	FALSE;
				ST_Complete				:=	FALSE;
				ST_Idle					:=	FALSE;
				ST_Held					:=	FALSE;
				ST_Suspended			:=	TRUE;
				ST_Stopped				:=	FALSE;
				ST_Aborted				:=	FALSE;
			END_IF
			
			IF Abort THEN
				ePMLState				:=	E_PMLState.ABORTING;
				ST_Suspended			:=	FALSE;
				ST_Aborting				:=	TRUE;
			ELSIF Stop THEN
				ePMLState				:=	E_PMLState.STOPPING;
				ST_Suspended			:=	FALSE;
				ST_Stopping				:=	TRUE;
			ELSIF UnSuspend THEN
				ePMLState				:=	E_PMLState.UNSUSPENDING;
				ST_Suspended			:=	FALSE;
				ST_UnSuspending			:=	TRUE;
			END_IF

		E_PMLState.UNSUSPENDING:	
			IF bStateChange	THEN
				ST_Starting				:=	FALSE;
				ST_Completing			:=	FALSE;
				ST_Resetting			:=	FALSE;
				ST_Holding				:=	FALSE;
				ST_UnHolding			:=	FALSE;
				ST_Suspending			:=	FALSE;
				ST_UnSuspending			:=	TRUE;
				ST_Clearing				:=	FALSE;
				ST_Stopping				:=	FALSE;
				ST_Aborting				:=	FALSE;
				
				ST_Execute				:=	FALSE;
				ST_Complete				:=	FALSE;
				ST_Idle					:=	FALSE;
				ST_Held					:=	FALSE;
				ST_Suspended			:=	FALSE;
				ST_Stopped				:=	FALSE;
				ST_Aborted				:=	FALSE;
			END_IF
			
			IF Abort THEN
				ePMLState				:=	E_PMLState.ABORTING;
				ST_UnSuspending			:=	FALSE;
				ST_Aborting				:=	TRUE;
			ELSIF Stop THEN
				ePMLState				:=	E_PMLState.STOPPING;
				ST_UnSuspending			:=	FALSE;
				ST_Stopping				:=	TRUE;
			ELSIF StateComplete AND NOT bStateCompletePrev THEN
				ePMLState				:=	E_PMLState.EXECUTE;
				bStateCompletePrev		:=	StateComplete;
				ST_UnSuspending			:=	FALSE;
				ST_Execute				:=	TRUE;								
			END_IF
		
		E_PMLState.STOPPING:
			IF bStateChange	THEN
				ST_Starting				:=	FALSE;
				ST_Completing			:=	FALSE;
				ST_Resetting			:=	FALSE;
				ST_Holding				:=	FALSE;
				ST_UnHolding			:=	FALSE;
				ST_Suspending			:=	FALSE;
				ST_UnSuspending			:=	FALSE;
				ST_Clearing				:=	FALSE;
				ST_Stopping				:=	TRUE;
				ST_Aborting				:=	FALSE;
				
				ST_Execute				:=	FALSE;
				ST_Complete				:=	FALSE;
				ST_Idle					:=	FALSE;
				ST_Held					:=	FALSE;
				ST_Suspended			:=	FALSE;
				ST_Stopped				:=	FALSE;
				ST_Aborted				:=	FALSE;
			END_IF
			
			IF Abort THEN
				ePMLState				:=	E_PMLState.ABORTING;
				ST_Stopping				:=	FALSE;
				ST_Aborting				:=	TRUE;
			ELSIF StateComplete AND NOT bStateCompletePrev THEN
				ePMLState				:=	E_PMLState.STOPPED;
				bStateCompletePrev		:=	StateComplete;
				ST_Stopping				:=	FALSE;
				ST_Stopped				:=	TRUE;								
			END_IF

		E_PMLState.STOPPED:
			IF bStateChange	THEN
				ST_Starting				:=	FALSE;
				ST_Completing			:=	FALSE;
				ST_Resetting			:=	FALSE;
				ST_Holding				:=	FALSE;
				ST_UnHolding			:=	FALSE;
				ST_Suspending			:=	FALSE;
				ST_UnSuspending			:=	FALSE;
				ST_Clearing				:=	FALSE;
				ST_Stopping				:=	FALSE;
				ST_Aborting				:=	FALSE;
				
				ST_Execute				:=	FALSE;
				ST_Complete				:=	FALSE;
				ST_Idle					:=	FALSE;
				ST_Held					:=	FALSE;
				ST_Suspended			:=	FALSE;
				ST_Stopped				:=	TRUE;
				ST_Aborted				:=	FALSE;
			END_IF
			
			IF Abort THEN
				ePMLState				:=	E_PMLState.ABORTING;
				ST_Stopped				:=	FALSE;
				ST_Aborting				:=	TRUE;
			ELSIF Reset THEN
				ePMLState				:=	E_PMLState.RESETTING;
				ST_Stopped				:=	FALSE;
				ST_Resetting			:=	TRUE;
			END_IF
		
		E_PMLState.ABORTING:
			IF bStateChange	THEN
				ST_Starting				:=	FALSE;
				ST_Completing			:=	FALSE;
				ST_Resetting			:=	FALSE;
				ST_Holding				:=	FALSE;
				ST_UnHolding			:=	FALSE;
				ST_Suspending			:=	FALSE;
				ST_UnSuspending			:=	FALSE;
				ST_Clearing				:=	FALSE;
				ST_Stopping				:=	FALSE;
				ST_Aborting				:=	TRUE;
				
				ST_Execute				:=	FALSE;
				ST_Complete				:=	FALSE;
				ST_Idle					:=	FALSE;
				ST_Held					:=	FALSE;
				ST_Suspended			:=	FALSE;
				ST_Stopped				:=	FALSE;
				ST_Aborted				:=	FALSE;
			END_IF
			
			IF StateComplete AND NOT bStateCompletePrev THEN
				ePMLState				:=	E_PMLState.ABORTED;
				bStateCompletePrev		:=	StateComplete;
				ST_Aborting				:=	FALSE;
				ST_Aborted				:=	TRUE;								
			END_IF
			
		E_PMLState.ABORTED:
			IF bStateChange	THEN
				ST_Starting				:=	FALSE;
				ST_Completing			:=	FALSE;
				ST_Resetting			:=	FALSE;
				ST_Holding				:=	FALSE;
				ST_UnHolding			:=	FALSE;
				ST_Suspending			:=	FALSE;
				ST_UnSuspending			:=	FALSE;
				ST_Clearing				:=	FALSE;
				ST_Stopping				:=	FALSE;
				ST_Aborting				:=	FALSE;
				
				ST_Execute				:=	FALSE;
				ST_Complete				:=	FALSE;
				ST_Idle					:=	FALSE;
				ST_Held					:=	FALSE;
				ST_Suspended			:=	FALSE;
				ST_Stopped				:=	FALSE;
				ST_Aborted				:=	TRUE;
			END_IF
			
			IF Clear THEN
				ePMLState				:=	E_PMLState.CLEARING;
				ST_Aborted				:=	FALSE;
				ST_Clearing				:=	TRUE;
			END_IF
		
		E_PMLState.CLEARING:
			IF bStateChange	THEN
				ST_Starting				:=	FALSE;
				ST_Completing			:=	FALSE;
				ST_Resetting			:=	FALSE;
				ST_Holding				:=	FALSE;
				ST_UnHolding			:=	FALSE;
				ST_Suspending			:=	FALSE;
				ST_UnSuspending			:=	FALSE;
				ST_Clearing				:=	TRUE;
				ST_Stopping				:=	FALSE;
				ST_Aborting				:=	FALSE;
				
				ST_Execute				:=	FALSE;
				ST_Complete				:=	FALSE;
				ST_Idle					:=	FALSE;
				ST_Held					:=	FALSE;
				ST_Suspended			:=	FALSE;
				ST_Stopped				:=	FALSE;
				ST_Aborted				:=	FALSE;
			END_IF
			
			IF Abort THEN
				ePMLState				:=	E_PMLState.ABORTING;
				ST_Clearing				:=	FALSE;
				ST_Aborting				:=	TRUE;
			ELSIF Stop THEN
				ePMLState				:=	E_PMLState.STOPPING;
				ST_Clearing				:=	FALSE;
				ST_Stopping				:=	TRUE;
			ELSIF StateComplete AND NOT bStateCompletePrev THEN
				ePMLState				:=	E_PMLState.STOPPED;
				bStateCompletePrev		:=	StateComplete;
				ST_Clearing				:=	FALSE;
				ST_Stopped				:=	TRUE;								
			END_IF
		
	END_CASE
	
	// bStateCompletePrev := bStateCompletePrev AND StateComplete;

END_FUNCTION_BLOCK

// ---- 00_Internal PackML/POUs/PS_PackML_UnitModeManager.TcPOU
FUNCTION_BLOCK PS_PackML_UnitModeManager
VAR_INPUT
	bExecute						:				BOOL;
	ePMLUnitModeCommand				:				E_PMLUnitMode;
	ePMLState						:				E_PMLState;
END_VAR
VAR_OUTPUT
	ePMLUnitModeStatus				:				E_PMLUnitMode;
	bDone							:				BOOL;
	bError							:				BOOL;
	nErrorID						:				UDINT;
END_VAR
VAR
	fbTriggerModeChange					:				R_TRIG;
END_VAR


	fbTriggerModeChange(CLK	:=	bExecute);

	IF fbTriggerModeChange.Q THEN
		bDone			:=		FALSE;
		bError			:=		FALSE;
		nErrorID		:=		0;
		
		CASE ePMLUnitModeStatus OF
			
			E_PMLUnitMode.UNDEFINED:
					ePMLUnitModeStatus	:=	ePMLUnitModeCommand;
					bDone				:=	TRUE;
			
			E_PMLUnitMode.AUTOMATIC:
					IF (ePMLState = E_PMLState.ABORTED) OR (ePMLState = E_PMLState.STOPPED) OR (ePMLState = E_PMLState.IDLE) THEN
						ePMLUnitModeStatus	:=	ePMLUnitModeCommand;
						bDone				:=	TRUE;
					ELSIF ((ePMLState = E_PMLState.HELD) OR (ePMLState = E_PMLState.SUSPENDED) OR (ePMLState = E_PMLState.COMPLETE))
						AND (ePMLUnitModeCommand = E_PMLUnitMode.SEMIAUTOMATIC) THEN
							ePMLUnitModeStatus	:=	ePMLUnitModeCommand;
							bDone				:=	TRUE;
					ELSIF (ePMLState = E_PMLState.HELD) AND (ePMLUnitModeCommand = E_PMLUnitMode.MAINTENANCE) THEN
							ePMLUnitModeStatus	:=	ePMLUnitModeCommand;
							bDone				:=	TRUE;
					ELSE
							bDone				:=	FALSE;
							bError				:=	TRUE;
							nErrorID			:=	1;
					END_IF
			E_PMLUnitMode.SEMIAUTOMATIC:
					IF (ePMLState = E_PMLState.ABORTED) OR (ePMLState = E_PMLState.STOPPED) OR (ePMLState = E_PMLState.IDLE) THEN
						ePMLUnitModeStatus	:=	ePMLUnitModeCommand;
						bDone				:=	TRUE;
					ELSIF ((ePMLState = E_PMLState.HELD) OR (ePMLState = E_PMLState.SUSPENDED) OR (ePMLState = E_PMLState.COMPLETE))
						AND (ePMLUnitModeCommand = E_PMLUnitMode.AUTOMATIC) THEN
							ePMLUnitModeStatus	:=	ePMLUnitModeCommand;
							bDone				:=	TRUE;
					ELSIF (ePMLState = E_PMLState.HELD) AND (ePMLUnitModeCommand = E_PMLUnitMode.MAINTENANCE) THEN
							ePMLUnitModeStatus	:=	ePMLUnitModeCommand;
							bDone				:=	TRUE;
					ELSE
							bDone				:=	FALSE;
							bError				:=	TRUE;
							nErrorID			:=	1;
					END_IF
			E_PMLUnitMode.MANUAL:
					IF (ePMLState = E_PMLState.ABORTED) OR (ePMLState = E_PMLState.STOPPED) OR (ePMLState = E_PMLState.IDLE) THEN
						ePMLUnitModeStatus	:=	ePMLUnitModeCommand;
						bDone				:=	TRUE;
					ELSE
							bDone				:=	FALSE;
							bError				:=	TRUE;
							nErrorID			:=	1;
					END_IF					
			E_PMLUnitMode.MAINTENANCE:
					IF (ePMLState = E_PMLState.ABORTED) OR (ePMLState = E_PMLState.STOPPED) OR (ePMLState = E_PMLState.IDLE) THEN
						ePMLUnitModeStatus	:=	ePMLUnitModeCommand;
						bDone				:=	TRUE;
					ELSIF (ePMLState = E_PMLState.HELD) AND ((ePMLUnitModeCommand = E_PMLUnitMode.AUTOMATIC) OR (ePMLUnitModeCommand = E_PMLUnitMode.SEMIAUTOMATIC)) THEN
							ePMLUnitModeStatus	:=	ePMLUnitModeCommand;
							bDone				:=	TRUE;
					ELSE
							bDone				:=	FALSE;
							bError				:=	TRUE;
							nErrorID			:=	1;
					END_IF					
					
			E_PMLUnitMode.DRYRUN:
					ePMLUnitModeStatus	:=	ePMLUnitModeCommand;
					bDone				:=	TRUE;
					
			E_PMLUnitMode.USERMODE1:
					ePMLUnitModeStatus	:=	ePMLUnitModeCommand;
					bDone				:=	TRUE;
					
			E_PMLUnitMode.USERMODE2:
					ePMLUnitModeStatus	:=	ePMLUnitModeCommand;
					bDone				:=	TRUE;
					
			E_PMLUnitMode.IDLE:
					IF (ePMLState = E_PMLState.ABORTED) OR (ePMLState = E_PMLState.STOPPED) OR (ePMLState = E_PMLState.IDLE) THEN
						ePMLUnitModeStatus	:=	ePMLUnitModeCommand;
						bDone				:=	TRUE;
					ELSE
							bDone				:=	FALSE;
							bError				:=	TRUE;
							nErrorID			:=	1;
					END_IF
			E_PMLUnitMode.ESTOP:
					IF (ePMLState = E_PMLState.ABORTED) OR (ePMLState = E_PMLState.STOPPED) OR (ePMLState = E_PMLState.IDLE) THEN
						ePMLUnitModeStatus	:=	ePMLUnitModeCommand;
						bDone				:=	TRUE;
					ELSE
							bDone				:=	FALSE;
							bError				:=	TRUE;
							nErrorID			:=	1;
					END_IF
		END_CASE
	END_IF

END_FUNCTION_BLOCK

// ---- 01_Submodules/Axis/FB_Axis.TcPOU
FUNCTION_BLOCK FB_Axis
VAR_OUTPUT
	bError			:	BOOL;				//Error signal
	nErrorID		:	UDINT;				//Error ID
	bMoving			:	BOOL;				// Status of moving
END_VAR
VAR
	bResetDone		:	BOOL;				// Status of function block MC_Reset
	bHaltDone		:	BOOL;				// Status of function block MC_Halt

	bStatusEnable	:	BOOL;				// Enable feedback
	
	fVelocity		:	LREAL;				// Target velocity
	fOverride		:	LREAL := 100;		// Override 100%
	
	fbTriggerHalt	:	R_TRIG;				// Trigger to recognize rising edge of halt input
	fbTriggerReset	:	R_TRIG;				// Trigger to recognize rising edge of reset input
	
	AxisRef			:	AXIS_REF;			// Axis reference (process data plc/nc)
	
	//=============== Motion function blocks =====================
	fbMcPower		:	MC_Power;			// FB for enable and override
	fbMcReset		:	MC_Reset;			// FB to reset axis (errors)
	fbMcStop		:	MC_Stop;				// FB to stop axis
	fbMcHalt		:	MC_Halt;				// FB to halt axis
	fbMcMove		:	Mc_MoveVelocity;	// FB to move axis (velocity movement)
	fbMcMoveAbsolute :	Mc_MoveAbsolute;	// FB to move axis (absolute position)
END_VAR

PROPERTY bState_Enable : BOOL
GET
bState_Enable := bStatusEnable;
END_GET
END_PROPERTY

PROPERTY bState_HaltDone : BOOL
GET
bState_HaltDone := bHaltDone;
END_GET
END_PROPERTY

PROPERTY bState_ResetDone : BOOL
GET
bState_ResetDone := bResetDone;
END_GET
END_PROPERTY

METHOD Enable
VAR_INPUT
	bEnable		:		BOOL;
END_VAR
fbMcPower(	Axis 			:= THIS^.AxisRef,
			Enable 			:=  bEnable,
			Enable_Positive := bEnable,
			Enable_Negative := bEnable,
			Override 		:= THIS^.fOverride,
			Status 			=> THIS^.bStatusEnable);
			
IF fbMcPower.Error THEN
	bError		:= TRUE;
	nErrorID	:= fbMcPower.ErrorID;
END_IF

AxisRef.ReadStatus();		// Axis internal method to read its status

THIS^.bMoving := AxisRef.Status.Moving;
END_METHOD

PROPERTY fTargetVelocity : LREAL
GET
fTargetVelocity := fVelocity;
END_GET
SET
fVelocity := fTargetVelocity;
END_SET
END_PROPERTY

METHOD Halt
VAR_INPUT
	bDriveHalt	:	BOOL;
END_VAR
// Move axis command set to FALSE
IF bDriveHalt THEN
	THIS^.fbMcMove( Axis 				:= THIS^.AxisRef,
					Execute 			:= FALSE);
	// ?? Move Absolute Execute FALSE ??
	THIS^.fbMcMoveAbsolute( Axis 		:= THIS^.AxisRef,
							Execute 	:= FALSE);		
ELSE
	THIS^.bHaltDone := FALSE;				
END_IF

//Trigger
THIS^.fbTriggerHalt(CLK := bDriveHalt);

IF THIS^.fbTriggerHalt.Q THEN
	THIS^.fbMcHalt( Axis			:= THIS^.AxisRef,
					Execute			:= TRUE);
ELSE
	THIS^.fbMcHalt( Axis			:= THIS^.AxisRef);
END_IF

// Done / Error / Aborted
IF THIS^.fbMcHalt.Done OR THIS^.fbMcHalt.Error OR THIS^.fbMcHalt.CommandAborted THEN
	THIS^.bError		:= THIS^.fbMcHalt.Error;
	THIS^.nErrorID		:= THIS^.fbMcHalt.ErrorID;
	THIS^.bHaltDone		:= THIS^.fbMcHalt.Done;

	THIS^.fbMcHalt( Axis 		:= THIS^.AxisRef,
					Execute		:= FALSE);
END_IF
END_METHOD

METHOD MoveBw
VAR_INPUT
END_VAR
IF NOT THIS^.fbMcMove.Error THEN
	fbMcMove(	Axis		:= THIS^.AxisRef,
				Execute		:= TRUE,
				Direction	:= MC_Negative_Direction,
				Velocity	:= THIS^.fVelocity);
END_IF

// Error / Command aborted
IF THIS^.fbMcMove.Error OR THIS^.fbMcMove.CommandAborted THEN
	THIS^.bError			:= THIS^.fbMcMove.Error;
	THIS^.nErrorID			:= THIS^.fbMcMove.ErrorID;
END_IF

	fbMcMove(	Axis		:= THIS^.AxisRef,
				Execute		:= FALSE);
END_METHOD

METHOD MoveFw
VAR_INPUT
END_VAR
IF NOT THIS^.fbMcMove.Error THEN
	fbMcMove(	Axis		:= THIS^.AxisRef,
				Execute		:= TRUE,
				Direction	:= MC_Positive_Direction,
				Velocity	:= THIS^.fVelocity);
END_IF

// Error / Command aborted
IF THIS^.fbMcMove.Error OR THIS^.fbMcMove.CommandAborted THEN
	THIS^.bError			:= THIS^.fbMcMove.Error;
	THIS^.nErrorID			:= THIS^.fbMcMove.ErrorID;
END_IF

	fbMcMove(	Axis		:= THIS^.AxisRef,
				Execute		:= FALSE);
END_METHOD

METHOD Reset
VAR_INPUT
	bDriveReset		:	BOOL;	// Request reset
END_VAR
IF NOT bDriveReset THEN
	THIS^.bResetDone := FALSE;
END_IF

// Trigger
THIS^.fbTriggerReset(CLK 		:= bDriveReset);

IF THIS^.fbTriggerReset.Q THEN
	THIS^.bResetDone := FALSE;
	THIS^.fbMcReset(Axis 		:= THIS^.AxisRef,
					Execute 	:= TRUE);
ELSE
	THIS^.fbMcReset(Axis 		:= THIS^.AxisRef);
END_IF

// Done / Error
IF THIS^.fbMcReset.Done OR THIS^.fbMcReset.Error THEN
	THIS^.bResetDone 			:= THIS^.fbMcReset.Done;
	THIS^.bError		 		:= THIS^.fbMcReset.Error;
	
	THIS^.fbMcReset (Axis 		:= THIS^.AxisRef,
					Execute 	:= FALSE);
END_IF
END_METHOD

METHOD Stop
VAR_INPUT
	bDriveStop	:	BOOL;		// Request drive stop
END_VAR
IF bDriveStop THEN
	// Move Execute FALSE
	THIS^.fbMcMove( Axis 				:= THIS^.AxisRef,
					Execute 			:= FALSE);			
	// ?? Move Absolute Execute FALSE ??
	THIS^.fbMcMoveAbsolute( Axis 		:= THIS^.AxisRef,
							Execute 	:= FALSE);			

ELSE
	THIS^.bHaltDone := FALSE;
END_IF

// Trigger
THIS^.fbTriggerHalt(CLK := bDriveStop);

IF fbTriggerHalt.Q THEN
	THIS^.fbMcStop( Axis 		:= THIS^.AxisRef,
					Execute 	:= TRUE);
END_IF

// Done / Error / Command aborted
IF THIS^.fbMcStop.Done OR THIS^.fbMcStop.Error OR THIS^.fbMcStop.CommandAborted THEN
	THIS^.bError				:= THIS^.fbMcStop.Error;
	THIS^.bError				:= THIS^.fbMcStop.Error;
	THIS^.bHaltDone				:= THIS^.fbMcStop.Done;
	
	THIS^.fbMcStop( Axis 		:= THIS^.AxisRef,
					Execute 	:= FALSE);
	
END_IF
END_METHOD

END_FUNCTION_BLOCK

// ---- 01_Submodules/Cylinder/FB_CylinderDiag.TcPOU
FUNCTION_BLOCK FB_CylinderDiag EXTENDS FB_CylinderBase
VAR_INPUT
	nTimeOut						:		TIME;			// Watchdog time for cylinder position monitoring
END_VAR
VAR_OUTPUT
	bError						:		BOOL;			// Error signal (derived from position watchdog)
	nErrorID					:		UDINT;			// Error ID
	sErrorMsg					:		STRING;			// Error Message
END_VAR
VAR
	fbTriggerError				:		R_TRIG;			// Trigger to recognize rising edge of error
	fbTimerWatchDog				:		TON;			// Watchdog timer for monitoring if cylinder reaches base/work position
END_VAR

// ============================================================
;
// ============================================================

METHOD Diag
VAR_INPUT
END_VAR
IF NOT bAtBasePos AND NOT bAtWorkPos THEN
	fbTimerWatchDog(	IN		:=		TRUE,
						PT		:=		nTimeOut);
ELSE
	fbTimerWatchDog(	IN		:=		FALSE,
						PT		:=		nTimeOut);
END_IF

	fbTriggerError(		CLK		:=		fbTimerWatchDog.Q);
	
	bError						:=		fbTimerWatchDog.Q;
	
IF bError	THEN
	IF	bMoveToWork		THEN
		sErrorMsg		:=		'Work position not reached';
		nErrorID		:=		92;
	ELSE
		sErrorMsg		:=		'Base position not reached';
		nErrorID		:=		91;
	END_IF
ELSE
	sErrorMsg			:=		'';
	nErrorID			:=		0;
END_IF
END_METHOD

METHOD Reset

// Calling Reset() method of parental class FB_Cylinder
SUPER^.Reset();

bError			:=		FALSE;
nErrorID		:=		0;
sErrorMsg		:=		'';
END_METHOD

METHOD PROTECTED StateMachine
VAR_INPUT
	bBasePosReq		:	BOOL;
	bWorkPosReq		:	BOOL;
END_VAR
IF NOT bError THEN
	// Calling StateMachine() method of parental class FB_Cylinder
	SUPER^.StateMachine(	bBasePosReq			:=		bBasePosReq,
							bWorkPosReq			:=		bWorkPosReq);
	
	// Diagnosis evaluation by every movement of cylinder							
	Diag();
END_IF
END_METHOD

END_FUNCTION_BLOCK

// ---- 01_Submodules/Cylinder/FB_CylinderBase.TcPOU
(* FB_Cylinder		- number of control signals:
							one direction is controllable
					- type of feedback:
							feedback is base and work position
*)

FUNCTION_BLOCK FB_CylinderBase IMPLEMENTS I_Cylinder
VAR_INPUT
	bAtBasePos		AT %I*		:	BOOL;		// Hardware input signal: cylinder is at base position
	bAtWorkPos		AT %I*		:	BOOL;		// Hardware input signal: cylinder is at work position
END_VAR
VAR_OUTPUT
	bMoveToWork		AT %Q*		:	BOOL;		// Hardware output signal to move cylinder to work position
END_VAR
VAR
END_VAR

// =================================================
;
// =================================================

{warning 'add property implementation'}
PROPERTY bState_AtBasePos : BOOL
GET
bState_AtBasePos := THIS^.bAtBasePos;
END_GET
END_PROPERTY

{warning 'add property implementation'}
PROPERTY bState_AtWorkPos : BOOL
GET
bState_AtWorkPos := THIS^.bAtWorkPos;
END_GET
END_PROPERTY

{warning 'add property implementation'}
PROPERTY bState_MoveToWork : BOOL
GET
bState_MoveToWork := THIS^.bMoveToWork;
END_GET
END_PROPERTY

METHOD MoveToBase
StateMachine(	bBasePosReq		:=		TRUE,
				bWorkPosReq		:=		FALSE);
END_METHOD

METHOD MoveToWork
StateMachine(	bBasePosReq		:=		FALSE,
				bWorkPosReq		:=		TRUE);
END_METHOD

METHOD Reset
THIS^.bMoveToWork		:=		FALSE;
END_METHOD

METHOD PROTECTED StateMachine
VAR_INPUT
	bBasePosReq		:	BOOL;
	bWorkPosReq		:	BOOL;
END_VAR
IF bWorkPosReq THEN
	THIS^.bMoveToWork 	:=		TRUE;
END_IF

IF bBasePosReq OR NOT bWorkPosReq THEN
	THIS^.bMoveToWork	:=		FALSE;
END_IF
END_METHOD

END_FUNCTION_BLOCK

// ---- 01_Submodules/Cylinder/FB_CylinderTemp.TcPOU
FUNCTION_BLOCK FB_CylinderTemp EXTENDS FB_CylinderBase
VAR_INPUT
	fTempCurrent		AT %I*		:		LREAL;		// Hardware input signal: cylinder temperature
END_VAR
VAR_OUTPUT
END_VAR
VAR
END_VAR

END_FUNCTION_BLOCK

// ---- 01_Submodules/Cylinder/FB_CylinderTempDiag.TcPOU
FUNCTION_BLOCK FB_CylinderTempDiag EXTENDS FB_CylinderTemp
VAR_INPUT
	fTempMin			:		LREAL;					// Global value:	minimal allowed cylinder temperature for temperature monitoring
	fTempMax			:		LREAL;					// Global value:	maximal allowed cylinder temperature for temperature monitoring
END_VAR
VAR_OUTPUT
	bError				:		BOOL;					// Error signal		(diagnosed from temperature monitoring)
	sErrorMsg			:		STRING;					// Error message
	nErrorID			:		UDINT;					// Error ID
END_VAR
VAR
END_VAR

METHOD Diag
VAR_INPUT
END_VAR
IF fTempCurrent > fTempMax OR fTempCurrent < fTempMin	THEN
	bError	:=	TRUE;
ELSE
	bError	:=	FALSE;
END_IF

IF bError	THEN
	IF		fTempCurrent > fTempMax	THEN
			sErrorMsg	:=		'Temperature above maximum';
			nErrorID	:=		94;
	ELSIF	fTempCurrent < fTempMin	THEN
			sErrorMsg	:=		'Temperature below minimum';
			nErrorID	:=		93;
	END_IF
ELSE
	sErrorMsg		:=	'';
	nErrorID		:=	0;
END_IF
END_METHOD

METHOD Reset
VAR_INPUT
END_VAR
SUPER^.Reset();

bError			:=		FALSE;
sErrorMsg		:=		'';
nErrorID		:=		0;
END_METHOD

METHOD PROTECTED StateMachine
VAR_INPUT
	bBasePosReq		:	BOOL;
	bWorkPosReq		:	BOOL;
END_VAR
IF NOT bError THEN
	// Calling StateMachine() method of parental class FB_Cylinder
	SUPER^.StateMachine(	bBasePosReq			:=		bBasePosReq,
							bWorkPosReq			:=		bWorkPosReq);
	
	// Diagnosis evaluation by every movement of cylinder							
	Diag();
END_IF
END_METHOD

END_FUNCTION_BLOCK

// ---- 01_Submodules/Cylinder/FB_CylinderTempRecord.TcPOU
FUNCTION_BLOCK FB_CylinderTempRecord EXTENDS FB_CylinderTemp
VAR_INPUT
	bRecordStart				:	BOOL;							// Signal to start recording temperature
	nTimeInterval				:	TIME;							// Time interval between samples of temperature
END_VAR
VAR_OUTPUT
	bRecordFullDone				:	BOOL;							// TRUE if the temperature recording is done
	aRecords					:	ARRAY [1..100] OF	LREAL;		//	Array with temperature records
END_VAR
VAR
	nIndex						:	UDINT;							// Index to handle temperature array
	fbTimerInterval				:	TON;							// Timer to control the recording interval
END_VAR

// ===================================================================
;
// ===================================================================

METHOD Record
VAR_INPUT
END_VAR

	bRecordFullDone := (nIndex := 100);

	IF bRecordStart AND NOT bRecordFullDone AND NOT fbTimerInterval.Q THEN
		fbTimerInterval(	IN		:=		TRUE,
							PT		:=		fbTimerInterval);
	END_IF
	
	IF fbTimerInterval.Q THEN
		fbTimerInterval(	IN		:=		FALSE);
		
		nIndex					:=		nIndex + 1;
		aRecords[nIndex]		:=		fTempCurrent;
	END_IF
END_METHOD

METHOD Reset
VAR_INPUT
END_VAR
	SUPER^.Reset();

	FOR nIndex	:= 1 TO 100 BY 1 DO
		aRecords[nIndex]	:=	0;
	END_FOR

	nIndex		:= 		0;
END_METHOD

END_FUNCTION_BLOCK

// ---- 02_Subsystems/FB_SeparatingModule.TcPOU
FUNCTION_BLOCK FB_SeparatingModule EXTENDS FB_SubsystemRoot
VAR_INPUT
	
	// ========================== State and mode of machine ==========================================================
	bExecute							:				BOOL;							// True in state EXECUTE
	bSemiStart							:				BOOL;							// Trigger for single process execution in semi-automatic mode

	nBoxOnConveyor						:				UINT;							// Actual number of boxes being processed
	
	// ========================== Button control for cylinders ======================================================================
	bButtonClampToWorkIn				:				BOOL;							// Signal from button to move clamp cylinder to work position
	bButtonClampToBaseIn				:				BOOL;							// Signal from button to move clamp cylinder to base position
	bButtonBarrierToWorkIn				:				BOOL;							// Signal from button to move barrier cylinder to work position
	bButtonBarrierToBaseIn				:				BOOL;							// Signal from button to move barrier cylinder to base position
	
END_VAR
VAR_OUTPUT
	bSeparated							:				BOOL;							// True if one separating process is done
	
	// ============================ Error variables =================================================================================
	bClampError							:				BOOL;							// Error signal of clamp cylinder
	sClampErrorMsg						:				STRING;							// Error message of clamp cylinder
	bBarrierError						:				BOOL;							// Error signal of barrier cylinder
	sBarrierErrorMsg					:				STRING;							// Error message of clamp cylinder
	
	// ============================= Temperature records =============================================================================
	aClampTemp							:				ARRAY[1..100] OF LREAL;			// Clamp cylinder temperature records
	aBarrierTemp						:				ARRAY[1..100] OF LREAL;			// Barrier cylinder temperature records
	
	// ========================== Button processed signal  ======================================================================
	bButtonClampToWorkOut				:				BOOL;							// Processed signal for button to move clamp cylinder to work position
	bButtonClampToBaseOut				:				BOOL;							// Processed signal for button to move clamp cylinder to base position
	bButtonBarrierToWorkOut				:				BOOL;							// Processed signal for button to move barrier cylinder to work position
	bButtonBarrierToBaseOut				:				BOOL;							// Processed signal for button to move barrier cylinder to base position
END_VAR
VAR
	// ========================== Function block instance of sensor ======================================================================
	fbSensor							:				FB_SignalHandlingIntern;		// Sensor for separting boxes process
	
	// ========================== Function block instance of clamp cylinder  ======================================================================
	fbClamp								:				FB_CylinderBase;					// Clamp cylinder without diagnosis and temperature records
	fbClampDiag							:				FB_CylinderDiag;					// Clamp cylinder with diagnosis
	fbClampTemp							:				FB_CylinderTemp;					// Clamp cylinder with temperature indication
	fbClampTempRecord					:				FB_CylinderTempRecord;				// Clamp cylinder with temperature record
	fbClampTempDiag						:				FB_CylinderTempDiag;				// Clamp cylinder with temperature diagnosis
	
	// ========================== Interface instance for clamp cylinder  ======================================================================
	itfClamp							:				I_Cylinder;							// Interface for flexible access to clamp cylinder FBs
	
	// ========================== Function block instance of barrier cylinder  ======================================================================
	fbBarrier							:				FB_CylinderBase;					// Barrier cylinder without diagnosis and temperature records
	fbBarrierDiag						:				FB_CylinderDiag;					// Barrier cylinder with diagnosis
	fbBarrierTemp						:				FB_CylinderTemp;					// Barrier cylinder with temperature indication
	fbBarrierTempRecord					:				FB_CylinderTempRecord;				// Barrier cylinder with temperature record
	fbBarrierTempDiag					:				FB_CylinderTempDiag;				// Barrier cylinder with temperature diagnosis
	
	// ========================== Interface instance for barrier cylinder  =============================================================================
	itfBarrier							:				I_Cylinder;							// Interface for flexible access to barrier cylinder FBs
	
	// ========================== Time parameters for clamp and barrier cylinder  ======================================================================
	tTimeOutClamp						:				TIME;								// For clamp cylinder with diagnosis: time in which the cylinder should reach base/work position
	tTimeOutBarrier						:				TIME;								// For barrier cylinder with diagnosis: time in which the cylinder should reach base/work position
	tTimeIntervalClamp					:				TIME;								// Time of intervals to record the temperature of clamp cylinder 
	tTimeIntervalBarrier				:				TIME;								// Time of intervals to record the temperature of barrier cylinder
	tTimeBarrierAtWork					:				TIME;								// Time period for separating process for which barrier cylinder stays at work position
	
	// ========================== Temperature parameters for clamp and barrier cylinder  ======================================================================
	nTempMinClamp						:				LREAL;								// For clamp cylinder with temperature diagnosis: minimal temperature
	nTempMinBarrier						:				LREAL;								// For barrier cylinder with temperature diagnosis: minimal temperature
	nTempMaxClamp						:				LREAL;								// For clamp cylinder with temperature diagnosis: maximal temperature
	nTempMaxBarrier						:				LREAL;								// For barrier cylinder with temperature diagnosis: maximal temperature
	
	// ============================ Signal handling for manual cylinders control  ======================================================================
	fbButtonClampToWork					:				FB_SignalHandlingIntern;			// Manual control of clamp cylinder to work position
	fbButtonClampToBase					:				FB_SignalHandlingIntern;			// Manual control of clamp cylinder to base position
	fbButtonBarrierToWork				:				FB_SignalHandlingIntern;			// Manual control of barrier cylinder to work position
	fbButtonBarrierToBase				:				FB_SignalHandlingIntern;			// Manual control of barrier cylinder to base position

	// ============================ Common variables ======================================================================
	fbTimerBarrierAtWork				:				TON;								// Timer for operning barrier in auto and semi-auto mode
	eStateAuto							:				E_StateSeparatingAutoClampBarrier;			// State variable for auto mode
	eStateSemiAuto						:				E_StateSeparatingAutoClampBarrier;			// State variable for semi-auto
	
END_VAR

// =========================================================
;
// =========================================================

METHOD Automatic
VAR_INPUT
END_VAR
	// Set timer delay for work position of barrier
	fbTimerBarrierAtWork(PT		:=		tTimeBarrierAtWork);
	
	IF NOT bHaltRequest	THEN
		fbAxis.MoveFw();
	
	ELSIF NOT bHaltDone THEN
		Stop(bStop	:= TRUE);
		
	ELSE
		Stop(bStop	:= FALSE);
	END_IF
	
// =========================================================
// State machine for process of separating boxes	
	
	CASE eStateAuto OF
		
		// =============================================================
		E_StateSeparatingAutoClampBarrier.Init:
		
						// Close clamp cylinder. Calling FB method through interface instance
						itfClamp.MoveToBase();
						
						// Checking if clamp is in initial position + execute active
						IF itfClamp.bState_AtBasePos AND bExecute THEN
							eStateAuto	:=	E_StateSeparatingAutoClampBarrier.Start;
						END_IF
		
		// =============================================================
		E_StateSeparatingAutoClampBarrier.Start:
		
						IF fbSensor.bOutputSignal AND fbAxis.bMoving THEN
							eStateAuto	:=	E_StateSeparatingAutoClampBarrier.CloseClamp;
						// Check if clamp cylinder is not opened
						ELSIF NOT	itfClamp.bState_AtWorkPos THEN
							itfClamp.MoveToWork();
						END_IF

		// =============================================================
		E_StateSeparatingAutoClampBarrier.CloseClamp:
		
						// Close clamp cylinder
						itfClamp.MoveToBase();
						
						// Check clamp cylinder closed and confirm separation bit
						IF itfClamp.bState_AtBasePos THEN
							bSeparated	:=	TRUE;
							eStateAuto	:=	E_StateSeparatingAutoClampBarrier.OpenBarrier;
						END_IF

		// =============================================================
		E_StateSeparatingAutoClampBarrier.OpenBarrier:
						
						// Open barrier cylinder
						itfBarrier.MoveToWork();

						// Check barrier cylinder closed
						IF itfBarrier.bState_AtWorkPos THEN
							fbTimerBarrierAtWork(IN	:= TRUE);
						END_IF

						IF fbTimerBarrierAtWork.Q THEN
							fbTimerBarrierAtWork(IN	:= FALSE);
							eStateAuto	:=	E_StateSeparatingAutoClampBarrier.CloseBarrier;
						END_IF
								
		// =============================================================
		E_StateSeparatingAutoClampBarrier.CloseBarrier:
		
						itfBarrier.MoveToBase();
						
						IF itfBarrier.bState_AtBasePos THEN
							bSeparated	:=	FALSE;
							eStateAuto	:=	E_StateSeparatingAutoClampBarrier.OpenClamp;	
						END_IF
		
		// =============================================================
		E_StateSeparatingAutoClampBarrier.OpenClamp:
		
						itfClamp.MoveToWork();
						
						IF itfClamp.bState_AtWorkPos THEN
							eStateAuto	:=	E_StateSeparatingAutoClampBarrier.Init;
						END_IF
												
		END_CASE
END_METHOD

PROPERTY bState_BarrierAtBasePos : BOOL
GET
END_GET
SET
END_SET
END_PROPERTY

PROPERTY bState_BarrierAtWorkPos : BOOL
GET
END_GET
SET
END_SET
END_PROPERTY

PROPERTY bState_ClampAtBasePos : BOOL
GET
END_GET
SET
END_SET
END_PROPERTY

PROPERTY bState_ClampAtWorkPos : BOOL
GET
END_GET
SET
END_SET
END_PROPERTY

METHOD CylinderOptions
VAR_INPUT
	bClampDiag					:				BOOL;			// If TRUE clamp cylinder has diagnostic functionality
	bClampTemp					:				BOOL;			// If TRUE clamp cylinder has temperature functionality
	bClampRecord				:				BOOL;			// If TRUE clamp cylinder has recording functionality	
	
	bBarrierDiag				:				BOOL;			// If TRUE barrier cylinder has diagnostic functionality
	bBarrierTemp				:				BOOL;			// If TRUE barrier cylinder has temperature functionality
	bBarrierRecord				:				BOOL;			// If TRUE barrier cylinder has recording functionality
END_VAR
	
	// Clamp cylinder interface
	
	IF bClampDiag THEN
		// Clamp cylinder with temperature diagnosis
		IF	bClampTemp THEN
			fbClampTempDiag.fTempMin				:=			nTempMinClamp;
			fbClampTempDiag.fTempMax				:=			nTempMaxClamp;
			bClampError								:=			fbClampTempDiag.bError;
			sClampErrorMsg							:=			fbClampTempDiag.sErrorMsg;
				itfClamp								:=			fbClampTempDiag;
		// Clamp cylinder with position diagnosis without temperature diagnosis
		ELSE
			bClampError								:=			fbClampDiag.bError;
			sClampErrorMsg							:=			fbClampDiag.sErrorMsg;
				itfClamp								:=			fbClampDiag;
		END_IF
	ELSE
		bClampError									:=			FALSE;
		sClampErrorMsg								:=			'';
		
		// Clamp cylinder with temperature record
		IF bClampTemp THEN
			IF bClampRecord THEN
				fbClampTempRecord.nTimeInterval		:=			tTimeIntervalClamp;				// Time of record intervals
				fbClampTempRecord.bRecordStart		:=			bCompresAirEnableLocal;			// Record if compressed air is set
				
				fbClampTempRecord.Record();														// Call record() method of FB_CylinderTempRecord
				
				aClampTemp							:=			fbClampTempRecord.aRecords;
					itfClamp							:=			fbClampTempRecord;
			ELSE
					itfClamp							:=			fbClampTemp;
			END_IF
		ELSE
					itfClamp							:=			fbClamp;
		END_IF
		
	END_IF
	
	// Barrier cylinder interface
	
	IF bBarrierDiag THEN
		IF	bBarrierTemp THEN
			fbBarrierTempDiag.fTempMin				:=			nTempMinBarrier;
			fbBarrierTempDiag.fTempMax				:=			ntempMaxBarrier;
			bBarrierError							:=			fbBarrierTempDiag.bError;
			sBarrierErrorMsg						:=			fbBarrierTempDiag.sErrorMsg;
				itfBarrier								:=			fbBarrierTempDiag;
		ELSE
			
			bBarrierError							:=			fbBarrierDiag.bError;
			sBarrierErrorMsg						:=			fbBarrierDiag.sErrorMsg;
				itfBarrier								:=			fbBarrierDiag;
		END_IF
	ELSE
		bBarrierError								:=			FALSE;
		sBarrierErrorMsg							:=			'';
		
		IF bBarrierTemp THEN
			IF bBarrierRecord THEN
				fbBarrierTempRecord.nTimeInterval	:=			tTimeIntervalBarrier;
				fbBarrierTempRecord.bRecordStart	:=			bCompresAirEnableLocal;
				
				fbBarrierTempRecord.Record();
				
				aBarrierTemp						:=			fbBarrierTempRecord.aRecords;
					itfBarrier							:=			fbBarrierTempRecord;
			ELSE
					itfBarrier							:=			fbBarrierTemp;
			END_IF
		ELSE
					itfBarrier							:=			fbBarrier;
		END_IF
		
	END_IF
END_METHOD

METHOD Enable
VAR_INPUT
	bComprAirEnable					:			BOOL;			// Enable of compressed air
	bAxisEnable						:			BOOL;			// Enable of axis
	bSensorEnable					:			BOOL;			// Enable of sensor
	bManualAxisEnable				:			BOOL;			// Enable manual axis control
END_VAR
	
	SUPER^.Enable(	bComprAirEnable		:=		bComprAirEnable,
					bAxisEnable			:=		bAxisEnable,
					bSensorEnable		:=		bSensorEnable,
					bManualAxisEnable	:=		bManualAxisEnable);
				
	// Sensor control
	
	fbSensor.Enable( bEnable			:=		bSensorEnable);
	
	// Clamp and barrier cylinder buttons control
	
	fbButtonClampToBase.Enable(		bEnable	:=		bManualCylinderEnableLocal AND NOT itfClamp.bState_AtBasePos);				// bManualAxisEnable + bComprAirEnable
	fbButtonClampToWork.Enable(		bEnable	:=		bManualCylinderEnableLocal AND NOT itfClamp.bState_AtWorkPos);
	
	fbButtonClampToBase.bInputSignal		:=		NOT fbButtonClampToWork.bInputSignal;
	
	fbButtonBarrierToBase.Enable(	bEnable	:=		bManualCylinderEnableLocal AND NOT itfBarrier.bState_AtBasePos);
	fbButtonBarrierToWork.Enable(	bEnable	:=		bManualCylinderEnableLocal AND NOT itfBarrier.bState_AtWorkPos);
	
	fbButtonBarrierToBase.bInputSignal		:=		NOT fbButtonBarrierToWork.bInputSignal;
END_METHOD

METHOD InputOutput
VAR_INPUT
END_VAR

	SUPER^.InputOutput();
	
	fbSensor.SetOutput();
	
	fbButtonClampToWork.SetOutput();
	fbButtonClampToBase.SetOutput();
	fbButtonBarrierToWork.SetOutput();
	fbButtonBarrierToWork.SetOutput();
	
	fbButtonClampToWork.bInputSignal					:=						bButtonClampToWorkIn;
	fbButtonClampToBase.bInputSignal					:=						bButtonClampToBaseIn;
	fbButtonBarrierToWork.bInputSignal					:=						bButtonBarrierToWorkIn;
	fbButtonBarrierToBase.bInputSignal					:=						bButtonBarrierToBaseIn;

	bButtonClampToWorkOut								:=						fbButtonClampToWork.bOutputSignal;
	bButtonClampToBaseOut								:=						fbButtonClampToBase.bOutputSignal;
	bButtonBarrierToWorkOut								:=						fbButtonBarrierToWork.bOutputSignal;
	bButtonBarrierToBaseOut								:=						fbButtonBarrierToBase.bOutputSignal;
END_METHOD

METHOD Maintain
VAR_INPUT
END_VAR

	THIS^.Manual();
END_METHOD

METHOD Manual
VAR_INPUT
END_VAR

	SUPER^.Manual();
	
	// Manual clamp & barrier cylinder control
	
	IF fbButtonClampToWork.bOutputSignal THEN
		itfClamp.MoveToWork();
	ELSIF	fbButtonClampToBase.bOutputSignal THEN
		itfClamp.MoveToBase();	
	END_IF
	
	IF fbButtonBarrierToWork.bOutputSignal THEN
		itfBarrier.MoveToWork();
	ELSIF	fbButtonBarrierToBase.bOutputSignal THEN
		itfBarrier.MoveToBase();
	END_IF
END_METHOD

PROPERTY nProp_TempMaxBarrier : LREAL
GET
nProp_TempMaxBarrier	:=	nTempMaxBarrier;
END_GET
SET
nTempMaxBarrier	:= nProp_TempMaxBarrier;
END_SET
END_PROPERTY

PROPERTY nProp_TempMaxClamp : LREAL
GET
nProp_TempMaxClamp	:=	nTempMaxClamp;
END_GET
SET
nTempMaxClamp	:=	nProp_TempMaxClamp;
END_SET
END_PROPERTY

PROPERTY nProp_TempMinBarrier : LREAL
GET
nProp_TempMinBarrier	:=	nTempMinBarrier;
END_GET
SET
nTempMinBarrier	:=	nProp_TempMinBarrier;
END_SET
END_PROPERTY

PROPERTY nProp_TempMinClamp : LREAL
GET
nProp_TempMinClamp	:=	nTempMinClamp;
END_GET
SET
nTempMinClamp	:=	nProp_TempMinClamp;
END_SET
END_PROPERTY

METHOD Reset
VAR_INPUT
	bReset				:			BOOL;			// True if machine is in state RESETTING
END_VAR

	SUPER^.Reset(bReset		:=		bReset);
	
	IF fbTriggerResetStart.Q THEN
		
		bExecute				:=				FALSE;
		
		bSeparated				:=				FALSE;
		
		fbTimerBarrierAtWork( IN:= FALSE);

		itfClamp.Reset();
		itfBarrier.Reset();
	END_IF
END_METHOD

METHOD ResetState
VAR_INPUT
END_VAR
// =========================================================
	eStateAuto					:=			E_StateSeparatingAutoClampBarrier.Init;
	eStateSemiAuto				:=			E_StateSeparatingAutoClampBarrier.Init;
// =========================================================
END_METHOD

METHOD Semiautomatic
VAR_INPUT
END_VAR
	// Set timer delay for work position of barrier
	fbTimerBarrierAtWork(PT		:=		tTimeBarrierAtWork);
	
	IF (nBoxOnConveyor = 0) AND (eStateSemiAuto = E_StateSeparatingAutoClampBarrier.Init) THEN
		Stop(bStop	:=	TRUE);
	END_IF
	
	IF NOT bHaltRequest	THEN
		fbAxis.MoveFw();
	
	ELSIF NOT bHaltDone THEN
		Stop(bStop	:= TRUE);
		
	ELSE
		Stop(bStop	:= FALSE);
	END_IF
	// =========================================================
// State machine for process of separating boxes	
	
	CASE eStateSemiAuto OF
		
		// =============================================================
		E_StateSeparatingAutoClampBarrier.Init:
		
						// Close clamp cylinder. Calling FB method through interface instance
						itfClamp.MoveToBase();
						
						// Checking if clamp is in initial position + execute active
						IF itfClamp.bState_AtBasePos AND bExecute AND bSemiStart THEN
							eStateSemiAuto	:=	E_StateSeparatingAutoClampBarrier.Start;
						END_IF
		
		// =============================================================
		E_StateSeparatingAutoClampBarrier.Start:
		
						IF fbSensor.bOutputSignal THEN
							eStateSemiAuto	:=	E_StateSeparatingAutoClampBarrier.CloseClamp;
						// Check if clamp cylinder is not opened
						ELSIF NOT	itfClamp.bState_AtWorkPos THEN
							itfClamp.MoveToWork();
							fbAxis.MoveFw();
						END_IF

		// =============================================================
		E_StateSeparatingAutoClampBarrier.CloseClamp:
		
						// Close clamp cylinder
						itfClamp.MoveToBase();
						
						// Check clamp cylinder closed and confirm separation bit
						IF itfClamp.bState_AtBasePos THEN
							bSeparated	:=	TRUE;
							eStateSemiAuto	:=	E_StateSeparatingAutoClampBarrier.OpenBarrier;
						END_IF

		// =============================================================
		E_StateSeparatingAutoClampBarrier.OpenBarrier:
						
						// Open barrier cylinder
						itfBarrier.MoveToWork();

						// Check barrier cylinder closed
						IF itfBarrier.bState_AtWorkPos THEN
							fbTimerBarrierAtWork(IN	:= TRUE);
						END_IF

						IF fbTimerBarrierAtWork.Q THEN
							fbTimerBarrierAtWork(IN	:= FALSE);
							eStateSemiAuto	:=	E_StateSeparatingAutoClampBarrier.CloseBarrier;
						END_IF
								
		// =============================================================
		E_StateSeparatingAutoClampBarrier.CloseBarrier:
		
						itfBarrier.MoveToBase();
						
						IF itfBarrier.bState_AtBasePos THEN
							bSeparated	:=	FALSE;
							eStateSemiAuto	:=	E_StateSeparatingAutoClampBarrier.OpenClamp;	
						END_IF
		
		// =============================================================
		E_StateSeparatingAutoClampBarrier.OpenClamp:
		
						itfClamp.MoveToWork();
						
						IF itfClamp.bState_AtWorkPos THEN
							eStateSemiAuto	:=	E_StateSeparatingAutoClampBarrier.Init;
						END_IF
												
		END_CASE
END_METHOD

PROPERTY tBarrierAtWorkPos : TIME
GET
END_GET
SET
END_SET
END_PROPERTY

PROPERTY tProp_TimeIntervalBarrier : TIME
GET
tProp_TimeIntervalBarrier	:=	tTimeIntervalBarrier;
END_GET
SET
tTimeIntervalBarrier	:=	tProp_TimeIntervalBarrier;
END_SET
END_PROPERTY

PROPERTY tProp_TimeIntervalClamp : TIME
GET
tProp_TimeIntervalClamp		:=	tTimeIntervalClamp;
END_GET
SET
tTimeIntervalClamp	:=	tProp_TimeIntervalClamp;
END_SET
END_PROPERTY

PROPERTY tProp_TimeOutBarrier : TIME
GET
END_GET
SET
END_SET
END_PROPERTY

PROPERTY tProp_TimeOutClamp : TIME
GET
END_GET
SET
END_SET
END_PROPERTY

END_FUNCTION_BLOCK

// ---- 02_Subsystems/FB_SubsystemRoot.TcPOU
// Base class of modules with AXIS and BUTTONS for manual control
FUNCTION_BLOCK FB_SubsystemRoot
VAR_INPUT
	bButtonAxisFwIn					:		BOOL;						// Signal of button to move axis forwards
	bButtonAxisBwIn					:		BOOL;						// Signal of button to move axis beckwards
END_VAR
VAR_OUTPUT
	bAxisError						:		BOOL;						// Error signal of axis
	nAxisErrorID					:		UDINT;						// Error ID of axis error
	
	bAxisMoves						:		BOOL;						// True if axis is moving
	
	bButtonAxisFwOut				:		BOOL;						// Processed signal from button to move axis forward 
	bButtonAxisBwOut				:		BOOL;						// Processed signal from button to move axis backward
END_VAR
VAR
	bHaltDone						:		BOOL;						// True if module is stopped
	bResetDone						:		BOOL;						// True if module is reseted
	bStartingDone					:		BOOL;						// True if module is started
	
	bCompresAirEnableLocal			:		BOOL;						// Enable of compressed air
	bAxisEnableLocal				:		BOOL;						// Enable of axis
	bSensorEnableLocal				:		BOOL;						// Enable of sensor
	bManualAxisEnableLocal			:		BOOL;						// Enable of manual axis control
	bManualCylinderEnableLocal		:		BOOL;						// Enable of manual cylinder control (not in the input of THIS^.Enable() )
	
	bHaltRequest					:		BOOL;						// True if machine is in state ABORTING or STOPPING
	bResetRequest					:		BOOL;						// True if machine is in state RESETTING
	
	// ============== Axis ========================================
	fbAxis							:		FB_Axis;					// Axis instance
	fAxisVelo						:		LREAL;						// Velocity of axis
	
	// ============ Manual axis control ==============================
	fbButtonAxisFw					:		FB_SignalHandlingIntern;	// Move axis forward
	fbButtonAxisBw					:		FB_SignalHandlingIntern;	// Move axis backward

